(* CODESYS project ProyectoAutomatasCodesys.project

Project tree, tasks and I/O mapping:
  Device : CODESYS Control Win V3, 3S - Smart Software Solutions GmbH, order no. 305021, version 3.5.9.20
    application Application
      libraries: Standard, * (System)
      task AutomataSeguridad (cyclic, interval t#100ms, priority 4) calls Nivel0
      task AutomataSupervisor (cyclic, interval t#50ms, priority 3) calls Nivel1
      task NivelControl (cyclic, interval t#22ms, priority 2) calls nivel2prueba
      task Planta (cyclic, interval t#1ms, priority 1) calls Planta
      task VISU_TASK (cyclic, interval 100 ms, priority 31) calls VisuElems.Visu_Prg
      program Nivel2 [ST]
      function block ControlAngulo [ST]
      function block Integrador [ST]
      function block Derivador [ST]
      program Nivel0 [SFC]: DuringRestaurarFuncionamiento, DuringFuncionamientoNormal, DuringEmergencia, DuringInit_RestaurarFuncionamiento, DuringDetenerCarro, DuringRegresarCarroNormalidad, DuringCarroDentroLimites, DuringDetenerIzaje, DuringRegresarIzajeNormalidad, DuringIzajeDentroLimites
      function block PIDCarro [ST]
      function block PIDIzaje [ST]
      Symbols
      global variables Global
      program Nivel1 [SFC]: tableroDeControl_active, grua_active, maquinaEspera_active, calculoSalidas_active, manual_active, manual_entry, manual_active_0, manual_entry_0, automatico_active, habilitaControlAngulo_active, habilitado_entry, deshabilitado_entry, gancho_active, Gabierto_entry, Gcerrado_entry, Gcerrado_active, pesoPermitido_entry, manualAuto_active, automatico_entry, pesoExcedido_entry, opManual_active, carro_active, izaje_active, verificacion_active, tableroActivo_entry, tableroActivo_active, tableroActivo_entry_0, tableroActivo_exit, limitesIzaje_active, dentroDeLimites_entry, cercaMinimo_entry, cercaMaximo_entry, cercaMaximo_active, manualAuto_entry, autoManual_active, autoManual_entry, start_active, actualizarParametros_active, start_entry, barcoAlMuelle_active, subirIzaje_entry, subirYdesplazarCarro_entry, Step0_barcoAlMuelle_active_entry, bajarYdesplazarCarro_entry, bajarCarro_entry, parar_entry, parar_active, parar_exit, subirIzaje_active, subirYdesplazarCarro_active, moverCarro_active, bajarYdesplazarCarro_active, bajarCarro_active, manualAuto_exit, autoManual_exit, cercaMinimo_active, subirYdesplazar_active, generador_active
      function AjusteGananciasCarro [ST]
      function block Saturation [ST]
      function block RateLimiter [ST]
      function AjusteBordesCarro [ST]
      program Planta [ST]
      function block Carro [ST]
      function block Izaje [ST]
      function block CargaSuspendida [ST]
      function block CableElastico [ST]
      function rectaDosPuntos [ST]
      function Transferencia [ST]
      function verificarChoquesLateralesMuelle [ST]
      function verificarChoquesLateralesBarco [ST]
      function trianguloDesaceleracion [ST]
      function trianguloAceleracion [ST]
      function round [ST]
      function block GeneradorDeTrayectorias [ST]
      function colisionMuelleAlBarcoDesacel [ST]
      function colisionMuelleAlBarcoAcel [ST]
      function colisionBarcoAlMuelleDesacel [ST]
      function colisionBarcoAlMuelleAcel [ST]
      function block determinarAlturasContenedores [ST]
      visualisation Visualization
      program nivel2prueba [ST]
  libraries: VisuSymbols, 3.5.10.0 (System)
  text list GlobalTextList
*)

// Device/Application/Global
VAR_GLOBAL
	//Con la planta
	xt: LREAL :=-30;
	lh: LREAL :=5;
	theta: LREAL :=0;
	ml: LREAL :=15000;
	Tt: LREAL :=0;
	Gcierre: BOOL :=0;
	Th: LREAL :=-15000*9.80665*0.75/30;
	
	//Con el tablero y mando
	
	BotonEmergencia: BOOL:= FALSE;
	BotonReset: BOOL:= FALSE;
	BotonAbrirGancho: BOOL:= FALSE;
	BotonCerrarGancho: BOOL:= FALSE;
	BotonOperarMaq: BOOL:= FALSE;
	BotonPararMaq: BOOL:= FALSE;
	BotonModoAutomatico: BOOL:= FALSE;
	BotonModoManual: BOOL:= FALSE;
	PalancaCarro: INT:= 0;
	PalancaIzaje: INT:= 0;
	BotonActivaControlAngulo: BOOL:= FALSE;
	BotonDesactivaControlAngulo: BOOL:= FALSE;
	
	//para el generador de trayectorias
	x_destino: LREAL:= -30;
	x_origen: LREAL:= -30;
	y_destino: LREAL:= 40;
	y_origen: LREAL:= 40;
	ySeguridadCarro: LREAL:= 40;
	PosicionCarroInicioDescensoIzaje: LREAL:= -999;
	alturaInicioDesplazamientoCarro: LREAL:= -999;
	contBarco: ARRAY[1..21, 1..13] OF LREAL;
	contMuelle: ARRAY[1..2, 1..7] OF LREAL;
	//Entre nivel 0 y 1
	
	DetenerNivel1: BOOL:= FALSE;
	
	//Entre nivel 0 y 2
	
	FuncionamientoIzaje: BOOL:= TRUE;
	FuncionamientoCarro: BOOL:= TRUE;
	ConsignaCarro: LREAL:= 0;
	ConsignaIzaje: LREAL:= 0;
	
	//Entre nivel 1 y 2
	
	vh: LREAL:= 0;	
	vt: LREAL:= 0;
	ControlAngulo: BOOL:= TRUE;
	ControlPos: BOOL:= FALSE;
	
	

	//constantes que se usan en los dos niveles de control
	amaxt: LREAL:= 1;
	vmaxt: LREAL:= 4;
	amaxh: LREAL:= 1;
	vmaxh: LREAL:= 3;
	dt_control: LREAL:=0.022;
	dt_planta: LREAL:=0.001;

	
END_VAR

// Device/Application/Nivel0
PROGRAM Nivel0
VAR
	IzajeListo: BOOL:= FALSE;
	CarroListo: BOOL:= FALSE;
END_VAR
VAR CONSTANT
	l_max_max_cable: LREAL:= 66;
	l_min_min_cable: LREAL:= 4;
	xt_max_max: LREAL:= 51;
	xt_min_min: LREAL:= -31;
	l_max_cable: LREAL:= 65;
	l_min_cable: LREAL:= 5;
	xt_max: LREAL:= 50;
	xt_min: LREAL:= -30;
	vmaxh: LREAL := 3;
	vmaxt: LREAL := 4;
END_VAR

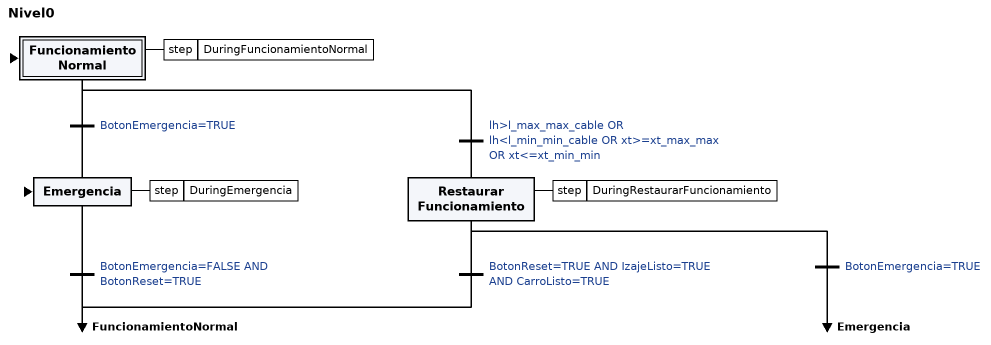
INITIAL_STEP FuncionamientoNormal:
    DuringFuncionamientoNormal(N);  // step action
END_STEP
TRANSITION FROM FuncionamientoNormal TO Emergencia
    := BotonEmergencia=TRUE;
END_TRANSITION
STEP Emergencia:
    DuringEmergencia(N);  // step action
END_STEP
TRANSITION FROM Emergencia TO FuncionamientoNormal
    := BotonEmergencia=FALSE AND BotonReset=TRUE;
END_TRANSITION
TRANSITION FROM FuncionamientoNormal TO RestaurarFuncionamiento
    := lh>l_max_max_cable OR lh<l_min_min_cable OR xt>=xt_max_max OR xt<=xt_min_min;
END_TRANSITION
STEP RestaurarFuncionamiento:
    DuringRestaurarFuncionamiento(N);  // step action
END_STEP
TRANSITION FROM RestaurarFuncionamiento TO FuncionamientoNormal
    := BotonReset=TRUE AND IzajeListo=TRUE AND CarroListo=TRUE;
END_TRANSITION
TRANSITION FROM RestaurarFuncionamiento TO Emergencia
    := BotonEmergencia=TRUE;
END_TRANSITION

ACTION DuringRestaurarFuncionamiento:
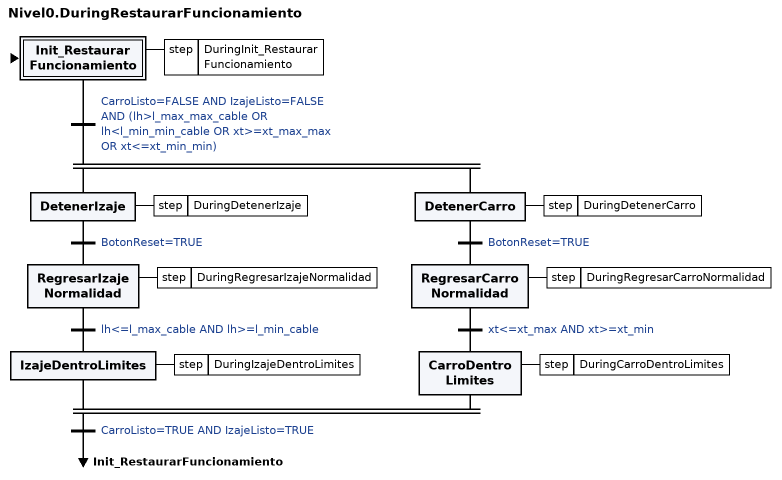
INITIAL_STEP Init_RestaurarFuncionamiento:
    DuringInit_RestaurarFuncionamiento(N);  // step action
END_STEP
TRANSITION FROM Init_RestaurarFuncionamiento TO (DetenerIzaje, DetenerCarro)
    := CarroListo=FALSE AND IzajeListo=FALSE AND (lh>l_max_max_cable OR lh<l_min_min_cable OR xt>=xt_max_max OR xt<=xt_min_min);
END_TRANSITION
STEP DetenerIzaje:
    DuringDetenerIzaje(N);  // step action
END_STEP
TRANSITION FROM DetenerIzaje TO RegresarIzajeNormalidad
    := BotonReset=TRUE;
END_TRANSITION
STEP RegresarIzajeNormalidad:
    DuringRegresarIzajeNormalidad(N);  // step action
END_STEP
TRANSITION FROM RegresarIzajeNormalidad TO IzajeDentroLimites
    := lh<=l_max_cable AND lh>=l_min_cable;
END_TRANSITION
STEP IzajeDentroLimites:
    DuringIzajeDentroLimites(N);  // step action
END_STEP
STEP DetenerCarro:
    DuringDetenerCarro(N);  // step action
END_STEP
TRANSITION FROM DetenerCarro TO RegresarCarroNormalidad
    := BotonReset=TRUE;
END_TRANSITION
STEP RegresarCarroNormalidad:
    DuringRegresarCarroNormalidad(N);  // step action
END_STEP
TRANSITION FROM RegresarCarroNormalidad TO CarroDentroLimites
    := xt<=xt_max AND xt>=xt_min;
END_TRANSITION
STEP CarroDentroLimites:
    DuringCarroDentroLimites(N);  // step action
END_STEP
TRANSITION FROM (IzajeDentroLimites, CarroDentroLimites) TO Init_RestaurarFuncionamiento
    := CarroListo=TRUE AND IzajeListo=TRUE;
END_TRANSITION
// branch label Branch0_RestaurarFuncionamiento
END_ACTION

ACTION DuringFuncionamientoNormal:
FuncionamientoIzaje:= TRUE;
FuncionamientoCarro:= TRUE;
DetenerNivel1:= FALSE;
END_ACTION

ACTION DuringEmergencia:
FuncionamientoIzaje:=FALSE;
FuncionamientoCarro:=FALSE;
ConsignaIzaje:=0;
ConsignaCarro:=0;
DetenerNivel1:=TRUE;
END_ACTION

ACTION DuringInit_RestaurarFuncionamiento:
IzajeListo:=FALSE;
CarroListo:=FALSE;
END_ACTION

ACTION DuringDetenerCarro:
IF (xt>=xt_max_max OR xt<=xt_min_min)
	THEN
	FuncionamientoCarro:= FALSE;
    ConsignaCarro:=0;
END_IF
END_ACTION

ACTION DuringRegresarCarroNormalidad:
DetenerNivel1:=TRUE;
FuncionamientoCarro:=FALSE;
IF (xt>xt_max)
	THEN
	ConsignaCarro:=-vmaxt/10;
END_IF
IF xt<xt_min
	THEN
    ConsignaCarro:=vmaxt/10;
END_IF
END_ACTION

ACTION DuringCarroDentroLimites:
CarroListo:=TRUE;
ConsignaCarro:=0;
END_ACTION

ACTION DuringDetenerIzaje:
IF (lh>l_max_max_cable OR lh<l_min_min_cable)
	THEN
	FuncionamientoIzaje:=FALSE;
    ConsignaIzaje:=0;
END_IF
END_ACTION

ACTION DuringRegresarIzajeNormalidad:
DetenerNivel1:= TRUE;
FuncionamientoIzaje:= FALSE;
IF (lh>l_max_cable)
	THEN
	ConsignaIzaje:=-vmaxh/10;
END_IF
IF (lh<l_min_cable)
	THEN
	ConsignaIzaje:=vmaxh/10;
END_IF
END_ACTION

ACTION DuringIzajeDentroLimites:
IzajeListo:=TRUE;
ConsignaIzaje:=0;
END_ACTION

END_PROGRAM

// Device/Application/Nivel1
PROGRAM Nivel1
VAR
	tiempoTableroActivo: LREAL:= 0;
	//tableroActivo:BOOL:=0;
	vhPermitidaIzq:LREAL:=0 ;
	vhPermitidaDer:LREAL:=0 ;
	finOperacion : BOOL:=1 ;
	vtmanual: LREAL := 0;
	vhmanual: LREAL := 0;
	
	vhauto: LREAL := 0;
	vtauto: LREAL := 0;
	
	x_destinoAnterior: LREAL :=999;
	Generador: GeneradorDeTrayectorias;
	
	tiempoTablero: ton ;
	tiempoManualAuto: ton ;
	tiempoModoAutomatico: ton;
	//para la transicion
	wait: ton;
	//Step: INT;
	
	//contadorTransicion: INT :=0;
	vmaxh: LREAL :=3;
	vmaxhfull: LREAL :=1.5;
	vmaxhSobrepeso: LREAL:=0.1;
	mlfull: LREAL := 65000;
	y_actual: LREAL := 45;
	//T: INT := 4;
	// auxiliar para manualAuto
	tiempo: LREAL := 0;
	cteAlturaInferior: LREAL;
	cteAlturaSuperior: LREAL;
	cteDestino: LREAL;
	n: INT := 0;
	veces: INT := 10;
	cteAlturaSuperior1: LREAL;
	cteCarro: LREAL;
END_VAR

VAR CONSTANT
	yt0: LREAL := 45;
	// se usa en limitesIzaje
	longitudSegMaxCable: LREAL := 60;
	longitudSegMinCable: LREAL := 10;
	l_max_cable: LREAL := 65;
	l_min_cable: LREAL := 5;
END_VAR

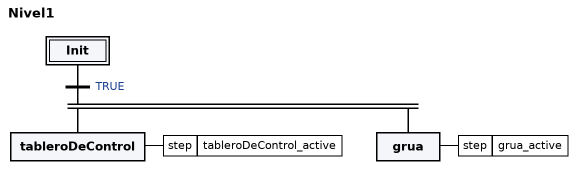
INITIAL_STEP Init:
END_STEP
TRANSITION FROM Init TO (tableroDeControl, grua)
    := TRUE;
END_TRANSITION
STEP tableroDeControl:
    tableroDeControl_active(N);  // step action
END_STEP
STEP grua:
    grua_active(N);  // step action
END_STEP

ACTION tableroDeControl_active:
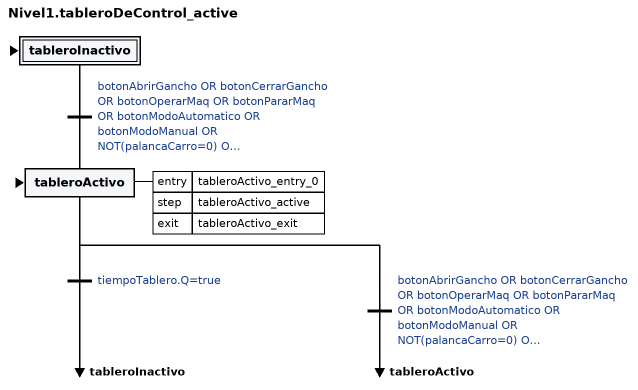
INITIAL_STEP tableroInactivo:
END_STEP
TRANSITION FROM tableroInactivo TO tableroActivo
    := botonAbrirGancho OR botonCerrarGancho OR botonOperarMaq OR botonPararMaq OR botonModoAutomatico OR botonModoManual OR NOT(palancaCarro=0) OR NOT(palancaIzaje=0);
END_TRANSITION
STEP tableroActivo:
    tableroActivo_entry_0(P1);  // entry action
    tableroActivo_active(N);  // step action
    tableroActivo_exit(P0);  // exit action
END_STEP
TRANSITION FROM tableroActivo TO tableroInactivo
    := tiempoTablero.Q=true;
END_TRANSITION
TRANSITION FROM tableroActivo TO tableroActivo
    := botonAbrirGancho OR botonCerrarGancho OR botonOperarMaq OR botonPararMaq OR botonModoAutomatico OR botonModoManual OR NOT(palancaCarro=0) OR NOT(palancaIzaje=0);
END_TRANSITION
// branch label Branch0_tableroDeControl_active
END_ACTION

ACTION grua_active:
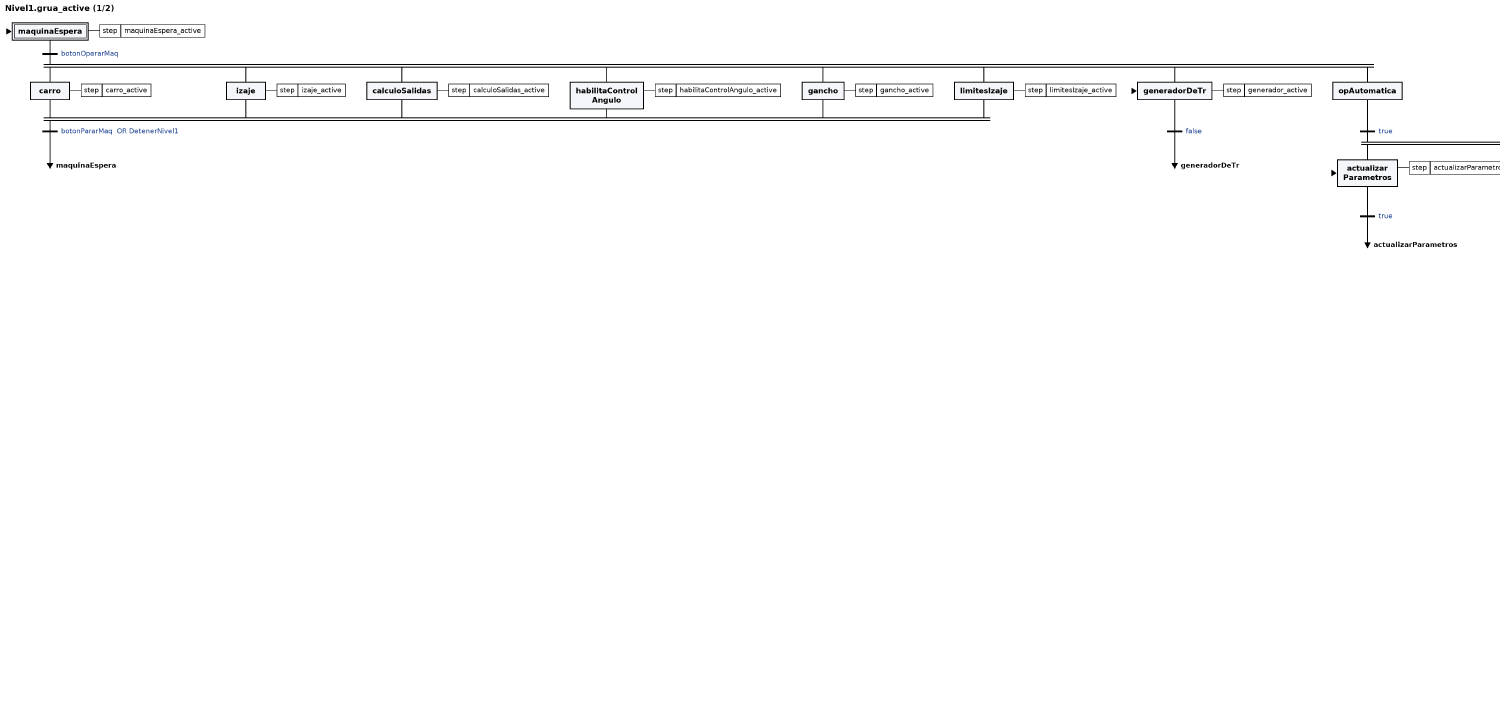
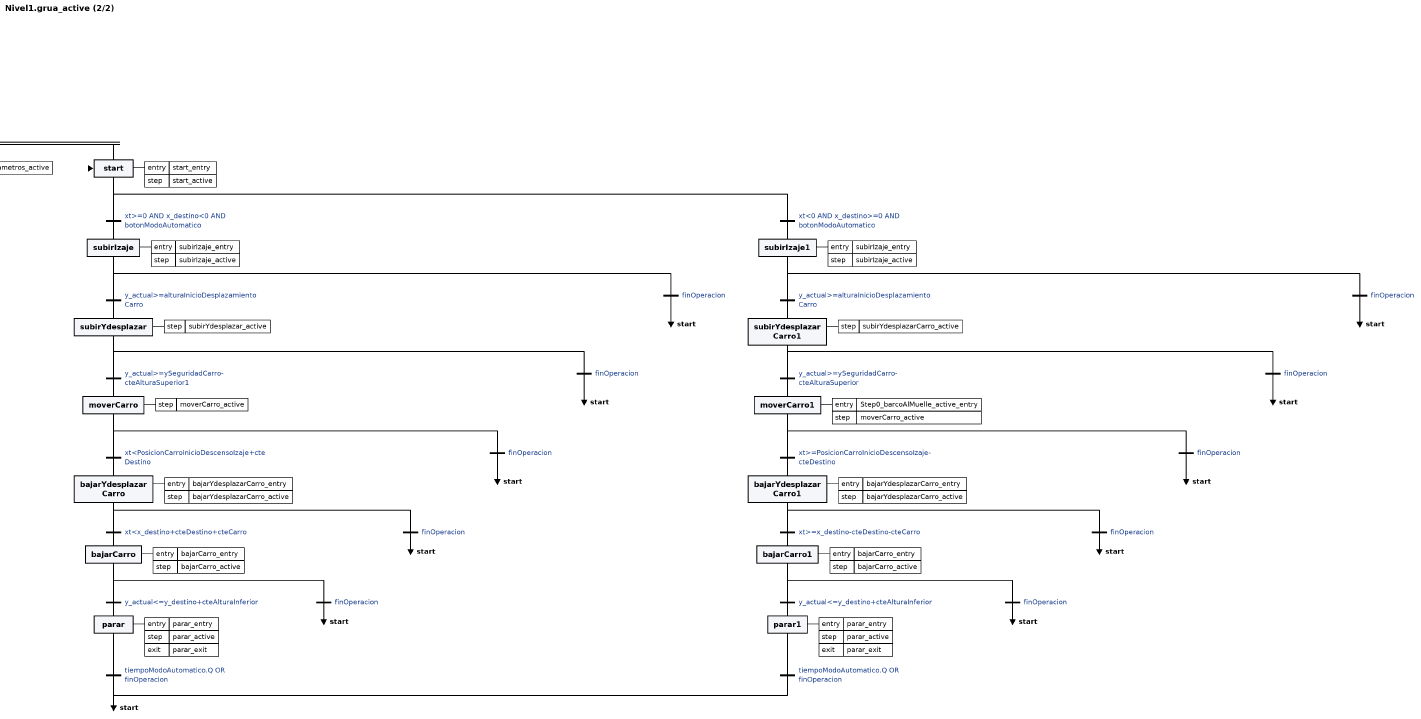
INITIAL_STEP maquinaEspera:
    maquinaEspera_active(N);  // step action
END_STEP
TRANSITION FROM maquinaEspera TO (carro, izaje, calculoSalidas, habilitaControlAngulo, gancho, limitesIzaje, generadorDeTr, opAutomatica)
    := botonOperarMaq;
END_TRANSITION
STEP carro:
    carro_active(N);  // step action
END_STEP
STEP izaje:
    izaje_active(N);  // step action
END_STEP
STEP calculoSalidas:
    calculoSalidas_active(N);  // step action
END_STEP
STEP habilitaControlAngulo:
    habilitaControlAngulo_active(N);  // step action
END_STEP
STEP gancho:
    gancho_active(N);  // step action
END_STEP
STEP limitesIzaje:
    limitesIzaje_active(N);  // step action
END_STEP
STEP generadorDeTr:
    generador_active(N);  // step action
END_STEP
TRANSITION FROM generadorDeTr TO generadorDeTr
    := false;
END_TRANSITION
STEP opAutomatica:
END_STEP
TRANSITION FROM opAutomatica TO (actualizarParametros, start)
    := true;
END_TRANSITION
STEP actualizarParametros:
    actualizarParametros_active(N);  // step action
END_STEP
TRANSITION FROM actualizarParametros TO actualizarParametros
    := true;
END_TRANSITION
STEP start:
    start_entry(P1);  // entry action
    start_active(N);  // step action
END_STEP
TRANSITION FROM start TO subirIzaje
    := xt>=0 AND x_destino<0 AND botonModoAutomatico;
END_TRANSITION
STEP subirIzaje:
    subirIzaje_entry(P1);  // entry action
    subirIzaje_active(N);  // step action
END_STEP
TRANSITION FROM subirIzaje TO subirYdesplazar
    := y_actual>=alturaInicioDesplazamientoCarro;
END_TRANSITION
STEP subirYdesplazar:
    subirYdesplazar_active(N);  // step action
END_STEP
TRANSITION FROM subirIzaje TO start
    := finOperacion;
END_TRANSITION
TRANSITION FROM subirYdesplazar TO moverCarro
    := y_actual>=ySeguridadCarro-cteAlturaSuperior1;
END_TRANSITION
TRANSITION FROM subirYdesplazar TO start
    := finOperacion;
END_TRANSITION
STEP moverCarro:
    moverCarro_active(N);  // step action
END_STEP
TRANSITION FROM moverCarro TO bajarYdesplazarCarro
    := xt<PosicionCarroInicioDescensoIzaje+cteDestino;
END_TRANSITION
TRANSITION FROM moverCarro TO start
    := finOperacion;
END_TRANSITION
STEP bajarYdesplazarCarro:
    bajarYdesplazarCarro_entry(P1);  // entry action
    bajarYdesplazarCarro_active(N);  // step action
END_STEP
TRANSITION FROM bajarYdesplazarCarro TO bajarCarro
    := xt<x_destino+cteDestino+cteCarro;
END_TRANSITION
TRANSITION FROM bajarYdesplazarCarro TO start
    := finOperacion;
END_TRANSITION
STEP bajarCarro:
    bajarCarro_entry(P1);  // entry action
    bajarCarro_active(N);  // step action
END_STEP
TRANSITION FROM bajarCarro TO parar
    := y_actual<=y_destino+cteAlturaInferior;
END_TRANSITION
TRANSITION FROM bajarCarro TO start
    := finOperacion;
END_TRANSITION
STEP parar:
    parar_entry(P1);  // entry action
    parar_active(N);  // step action
    parar_exit(P0);  // exit action
END_STEP
TRANSITION FROM parar TO start
    := tiempoModoAutomatico.Q OR finOperacion;
END_TRANSITION
TRANSITION FROM start TO subirIzaje1
    := xt<0 AND x_destino>=0 AND botonModoAutomatico;
END_TRANSITION
STEP subirIzaje1:
    subirIzaje_entry(P1);  // entry action
    subirIzaje_active(N);  // step action
END_STEP
TRANSITION FROM subirIzaje1 TO subirYdesplazarCarro1
    := y_actual>=alturaInicioDesplazamientoCarro;
END_TRANSITION
TRANSITION FROM subirIzaje1 TO start
    := finOperacion;
END_TRANSITION
STEP subirYdesplazarCarro1:
    subirYdesplazarCarro_active(N);  // step action
END_STEP
TRANSITION FROM subirYdesplazarCarro1 TO moverCarro1
    := y_actual>=ySeguridadCarro-cteAlturaSuperior;
END_TRANSITION
TRANSITION FROM subirYdesplazarCarro1 TO start
    := finOperacion;
END_TRANSITION
STEP moverCarro1:
    Step0_barcoAlMuelle_active_entry(P1);  // entry action
    moverCarro_active(N);  // step action
END_STEP
TRANSITION FROM moverCarro1 TO bajarYdesplazarCarro1
    := xt>=PosicionCarroInicioDescensoIzaje-cteDestino;
END_TRANSITION
TRANSITION FROM moverCarro1 TO start
    := finOperacion;
END_TRANSITION
STEP bajarYdesplazarCarro1:
    bajarYdesplazarCarro_entry(P1);  // entry action
    bajarYdesplazarCarro_active(N);  // step action
END_STEP
TRANSITION FROM bajarYdesplazarCarro1 TO bajarCarro1
    := xt>=x_destino-cteDestino-cteCarro;
END_TRANSITION
TRANSITION FROM bajarYdesplazarCarro1 TO start
    := finOperacion;
END_TRANSITION
STEP bajarCarro1:
    bajarCarro_entry(P1);  // entry action
    bajarCarro_active(N);  // step action
END_STEP
TRANSITION FROM bajarCarro1 TO parar1
    := y_actual<=y_destino+cteAlturaInferior;
END_TRANSITION
TRANSITION FROM bajarCarro1 TO start
    := finOperacion;
END_TRANSITION
STEP parar1:
    parar_entry(P1);  // entry action
    parar_active(N);  // step action
    parar_exit(P0);  // exit action
END_STEP
TRANSITION FROM parar1 TO start
    := tiempoModoAutomatico.Q OR finOperacion;
END_TRANSITION
TRANSITION FROM (carro, izaje, calculoSalidas, habilitaControlAngulo, gancho, limitesIzaje) TO maquinaEspera
    := botonPararMaq OR DetenerNivel1;
END_TRANSITION
// branch label Branch3_grua_active
// branch label Branch4_grua_active
// branch label Branch5_grua_active
// branch label Branch6_grua_active
// branch label Branch7_grua_active
// branch label Branch2_grua_active
// branch label Branch1_grua_active
// branch label Branch0_maquinaOperando_active
END_ACTION

ACTION maquinaEspera_active:
vt:=0;
vh:=0;
vhPermitidaIzq:=0 ;
vhPermitidaDer:=0 ;
END_ACTION

ACTION calculoSalidas_active:
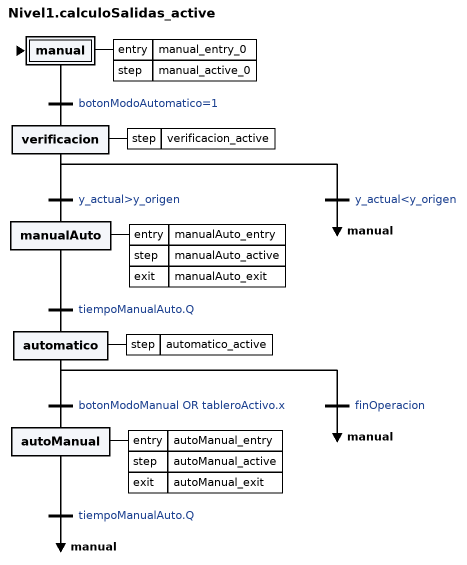
INITIAL_STEP manual:
    manual_entry_0(P1);  // entry action
    manual_active_0(N);  // step action
END_STEP
TRANSITION FROM manual TO verificacion
    := botonModoAutomatico=1;
END_TRANSITION
STEP verificacion:
    verificacion_active(N);  // step action
END_STEP
TRANSITION FROM verificacion TO manualAuto
    := y_actual>y_origen;
END_TRANSITION
TRANSITION FROM verificacion TO manual
    := y_actual<y_origen;
END_TRANSITION
STEP manualAuto:
    manualAuto_entry(P1);  // entry action
    manualAuto_active(N);  // step action
    manualAuto_exit(P0);  // exit action
END_STEP
TRANSITION FROM manualAuto TO automatico
    := tiempoManualAuto.Q;
END_TRANSITION
STEP automatico:
    automatico_active(N);  // step action
END_STEP
TRANSITION FROM automatico TO autoManual
    := botonModoManual OR tableroActivo.x;
END_TRANSITION
TRANSITION FROM automatico TO manual
    := finOperacion;
END_TRANSITION
STEP autoManual:
    autoManual_entry(P1);  // entry action
    autoManual_active(N);  // step action
    autoManual_exit(P0);  // exit action
END_STEP
TRANSITION FROM autoManual TO manual
    := tiempoManualAuto.Q;
END_TRANSITION
// branch label Branch0_calculoSalidas_active
// branch label Branch1_calculoSalidas_active
END_ACTION

ACTION manual_active:

END_ACTION

ACTION manual_entry:
controlPos :=0;
finOperacion :=1;
END_ACTION

ACTION manual_active_0:
vt :=vtmanual;
vh :=vhmanual;
END_ACTION

ACTION manual_entry_0:
controlPos :=0;
finOperacion :=1;
tiempoManualAuto.IN  :=0;
END_ACTION

ACTION automatico_active:
vt:=vtauto;
vh:=vhauto;
END_ACTION

ACTION habilitaControlAngulo_active:
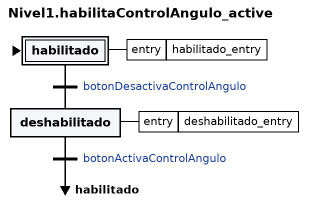
INITIAL_STEP habilitado:
    habilitado_entry(P1);  // entry action
END_STEP
TRANSITION FROM habilitado TO deshabilitado
    := botonDesactivaControlAngulo;
END_TRANSITION
STEP deshabilitado:
    deshabilitado_entry(P1);  // entry action
END_STEP
TRANSITION FROM deshabilitado TO habilitado
    := botonActivaControlAngulo;
END_TRANSITION
END_ACTION

ACTION habilitado_entry:
controlAngulo:=1;
END_ACTION

ACTION deshabilitado_entry:
controlAngulo:=0;
END_ACTION

ACTION gancho_active:
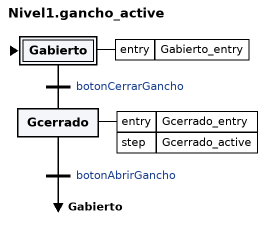
INITIAL_STEP Gabierto:
    Gabierto_entry(P1);  // entry action
END_STEP
TRANSITION FROM Gabierto TO Gcerrado
    := botonCerrarGancho;
END_TRANSITION
STEP Gcerrado:
    Gcerrado_entry(P1);  // entry action
    Gcerrado_active(N);  // step action
END_STEP
TRANSITION FROM Gcerrado TO Gabierto
    := botonAbrirGancho;
END_TRANSITION
END_ACTION

ACTION Gabierto_entry:
Gcierre:=0;
vhPermitidaIzq:=vmaxh;
vhPermitidaDer:= vmaxh;
END_ACTION

ACTION Gcerrado_entry:
Gcierre:=1;
END_ACTION

ACTION Gcerrado_active:
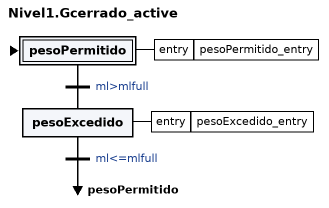
INITIAL_STEP pesoPermitido:
    pesoPermitido_entry(P1);  // entry action
END_STEP
TRANSITION FROM pesoPermitido TO pesoExcedido
    := ml>mlfull;
END_TRANSITION
STEP pesoExcedido:
    pesoExcedido_entry(P1);  // entry action
END_STEP
TRANSITION FROM pesoExcedido TO pesoPermitido
    := ml<=mlfull;
END_TRANSITION
END_ACTION

ACTION pesoPermitido_entry:
vhPermitidaIzq :=vmaxhfull ;
vhPermitidaDer:=vmaxhfull ;
END_ACTION

ACTION manualAuto_active:
tiempoManualAuto();
tiempo:=TIME_TO_LREAL(tiempoManualAuto.ET)/1000;
Transferencia(1.0,tiempo,vtmanual,vtauto,vhmanual,vhauto,Vh=>vh,Vt=>vt);
END_ACTION

ACTION automatico_entry:

END_ACTION

ACTION pesoExcedido_entry:
vhPermitidaIzq :=vmaxhSobrepeso ;
vhPermitidaDer:=vmaxhSobrepeso ;
END_ACTION

ACTION opManual_active:
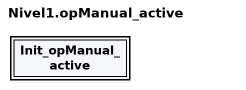
INITIAL_STEP Init_opManual_active:
END_STEP
END_ACTION

ACTION carro_active:
IF palancaCarro=-1 THEN
    vtmanual:=-vmaxt;
ELSIF palancaCarro=0 THEN
    vtmanual:=0; 
ELSIF palancaCarro=1 THEN
    vtmanual:=vmaxt;
END_IF
END_ACTION

ACTION izaje_active:
IF palancaIzaje=1 THEN
    vhmanual := vhPermitidaIzq;
ELSIF palancaIzaje=0 THEN
    vhmanual := 0;
ELSIF palancaIzaje=-1 THEN
    vhmanual := -vhPermitidaDer;
END_IF
END_ACTION

ACTION verificacion_active:
y_actual:=yt0-lh;
END_ACTION

ACTION tableroActivo_entry:
tiempoTablero(IN:=0,PT:=T#4S);
tiempoTablero.IN  :=1;
END_ACTION

ACTION tableroActivo_active:
tiempoTablero();
END_ACTION

ACTION tableroActivo_entry_0:
tiempoTablero.IN  :=0;
tiempoTablero(IN:=1,PT:=T#1S);
END_ACTION

ACTION tableroActivo_exit:
tiempoTablero(IN:=0);
END_ACTION

ACTION limitesIzaje_active:
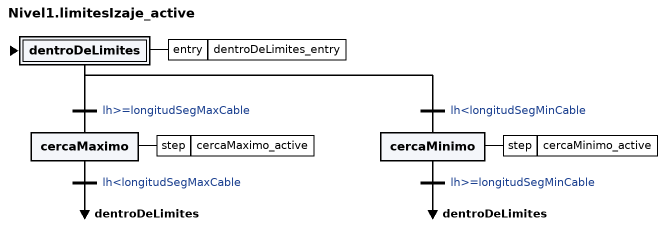
INITIAL_STEP dentroDeLimites:
    dentroDeLimites_entry(P1);  // entry action
END_STEP
TRANSITION FROM dentroDeLimites TO cercaMaximo
    := lh>=longitudSegMaxCable;
END_TRANSITION
STEP cercaMaximo:
    cercaMaximo_active(N);  // step action
END_STEP
TRANSITION FROM cercaMaximo TO dentroDeLimites
    := lh<longitudSegMaxCable;
END_TRANSITION
TRANSITION FROM dentroDeLimites TO cercaMinimo
    := lh<longitudSegMinCable;
END_TRANSITION
STEP cercaMinimo:
    cercaMinimo_active(N);  // step action
END_STEP
TRANSITION FROM cercaMinimo TO dentroDeLimites
    := lh>=longitudSegMinCable;
END_TRANSITION
// branch label Branch0_limitesIzaje_active
END_ACTION

ACTION dentroDeLimites_entry:
IF Gcierre THEN
	vhPermitidaIzq:= vmaxhfull;
	vhPermitidaDer:=vmaxhfull;
	
ELSE
	vhPermitidaIzq:=vmaxh ;
	vhPermitidaDer:=vmaxh ;
END_IF
END_ACTION

ACTION cercaMinimo_entry:

END_ACTION

ACTION cercaMaximo_entry:

END_ACTION

ACTION cercaMaximo_active:
IF Gcierre THEN
    vhPermitidaIzq:=rectaDosPuntos(vmaxh  ,0,longitudSegMaxCable,l_max_cable,lh);
else
    vhPermitidaIzq:=rectaDosPuntos(vmaxhfull,0,longitudSegMaxCable,l_max_cable,lh);
END_IF
END_ACTION

ACTION manualAuto_entry:
tiempoManualAuto.IN  :=0;
tiempoManualAuto(IN:=1,PT:=T#5S);
END_ACTION

ACTION autoManual_active:
tiempoManualAuto();
tiempo:=TIME_TO_LREAL(tiempoManualAuto.ET);
Transferencia(-1.0,tiempo,vtmanual,vtauto,vhmanual,vhauto);
END_ACTION

ACTION autoManual_entry:
tiempoManualAuto.IN  :=0;
tiempoManualAuto(IN:=1,PT:=T#5S);
END_ACTION

ACTION start_active:
y_actual:=yt0-lh;
END_ACTION

ACTION actualizarParametros_active:
 IF lh<22 THEN
     IF Gcierre THEN
         cteAlturaInferior:=6;
         cteAlturaSuperior:=-2;
         cteDestino:=0;
		 cteCarro:=10;
     else
         cteAlturaInferior:=6;
         cteAlturaSuperior:=10;
         cteDestino:=5;
		 cteCarro:=10;
     END_IF
 else
     IF Gcierre THEN
		 cteAlturaSuperior1:=2;
         cteAlturaInferior:=9;
         cteAlturaSuperior:=-2;
         cteDestino:=0;
		 cteCarro:=12;
     ELSE
		 cteAlturaSuperior1:=2;
         cteAlturaInferior:=10;
         cteAlturaSuperior:=4;
         cteDestino:=6;
		 cteCarro:=12;
     END_IF
 END_IF
END_ACTION

ACTION start_entry:
finOperacion:=0;
vtauto:=0;
vhauto:=0;
END_ACTION

ACTION barcoAlMuelle_active:
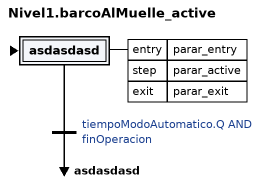
INITIAL_STEP asdasdasd:
    parar_entry(P1);  // entry action
    parar_active(N);  // step action
    parar_exit(P0);  // exit action
END_STEP
TRANSITION FROM asdasdasd TO asdasdasd
    := tiempoModoAutomatico.Q AND finOperacion;
END_TRANSITION
END_ACTION

ACTION subirIzaje_entry:

END_ACTION

ACTION subirYdesplazarCarro_entry:

END_ACTION

ACTION Step0_barcoAlMuelle_active_entry:

END_ACTION

ACTION bajarYdesplazarCarro_entry:
vhauto:=vhPermitidaIzq;
controlPos :=1;
END_ACTION

ACTION bajarCarro_entry:
vtauto:=0;
END_ACTION

ACTION parar_entry:
vhauto:=0;
tiempoModoAutomatico.IN  :=0;
tiempoModoAutomatico(IN:=1,PT:=T#60S);
END_ACTION

ACTION parar_active:
tiempoModoAutomatico();
y_actual:=yt0-lh;
END_ACTION

ACTION parar_exit:
tiempoModoAutomatico.IN  :=0;
finOperacion:=1;
END_ACTION

ACTION subirIzaje_active:
y_actual:=yt0-lh;
vhauto:=-vhPermitidaDer;
END_ACTION

ACTION subirYdesplazarCarro_active:
y_actual:=yt0-lh;
vtauto:=vmaxt;
END_ACTION

ACTION moverCarro_active:
y_actual:=yt0-lh;
vhauto:=0;
END_ACTION

ACTION bajarYdesplazarCarro_active:
y_actual:=yt0-lh;
END_ACTION

ACTION bajarCarro_active:
y_actual:=yt0-lh;
END_ACTION

ACTION manualAuto_exit:
tiempoManualAuto(IN  :=0, PT:=t#10s);
END_ACTION

ACTION autoManual_exit:
tiempoManualAuto(IN  :=0, PT:=t#10s);
END_ACTION

ACTION cercaMinimo_active:
IF Gcierre THEN
    vhPermitidaDer:=rectaDosPuntos(vmaxhfull,0,longitudSegMinCable,l_min_cable,lh);
else
    vhPermitidaDer:=rectaDosPuntos(vmaxh ,0,longitudSegMinCable,l_min_cable,lh);
END_IF
END_ACTION

ACTION subirYdesplazar_active:
y_actual:=yt0-lh;
vtauto:=-vmaxt;
END_ACTION

ACTION generador_active:
IF NOT (x_destinoAnterior=x_destino)
	THEN
	Generador();
	x_destinoAnterior:=x_destino;
END_IF
END_ACTION

END_PROGRAM

// Device/Application/GeneradorDeTrayectorias
FUNCTION_BLOCK GeneradorDeTrayectorias
VAR_INPUT
END_VAR
VAR_OUTPUT
END_VAR
VAR
	vIzaje: LREAL;
	alturaInicioAutomatico: LREAL;
	cantContDeSeguridad: LREAL;
	vCarro: LREAL;
	aTriangulo: LREAL;
	bTriangulo: LREAL;
	cTriangulo: LREAL;
	betaTriangulo: LREAL;
	determinarAlturasContenedores1: determinarAlturasContenedores;
	alturasContMuelle: ARRAY [1..7] OF LREAL;
	alturasContBarco: ARRAY [1..13] OF LREAL;
	nroColOrigen: INT;
	nroColDestino: INT;
	cuantosCont: LREAL;
	i: INT;
	donde: LREAL;
END_VAR
VAR CONSTANT
	vmaxh: LREAL:= 3;
	vmaxhfull: LREAL:= 1.5;
	vmaxt: LREAL:= 4;
	altoCont: LREAL:= 2.591;
	y_min: LREAL:=-20;
	xt_min: LREAL:= -30;
	divHoriz: LREAL:= 3.438;
	nroHorizContMuelle: INT:= 7;
	altoVigaTestera: LREAL:= 15;
	nroHorizContBarco: INT:=13;
END_VAR

//obtener posicion actual del carro
x_origen:=xt;
IF (Gcierre=1)
	THEN
    vIzaje:=vmaxhfull;
    alturaInicioAutomatico := altoCont * 1.5;
    cantContDeSeguridad:=2;
ELSE
    vIzaje:=vmaxh;
    alturaInicioAutomatico := altoCont * 0.5;
    cantContDeSeguridad:=1;
END_IF
vCarro:=vmaxt;
//calculo del triangulo de velocidades para las trayectorias
aTriangulo:=vCarro;
bTriangulo:=vIzaje;
cTriangulo:=SQRT(EXPT(aTriangulo,2)+EXPT(bTriangulo,2)); //hipotenusa
betaTriangulo:=ACOS(bTriangulo/cTriangulo);

y_destino:=999;
//inicialiar las variables, deben ser numeros negativos!!!!!!!
alturaInicioDesplazamientoCarro:=-999;
PosicionCarroInicioDescensoIzaje:=-999;
ySeguridadCarro:=-999;
//altura de seguridad para evitar colision entre el contenedor suspendido y
//las columnas de contenedores apilados. si este valor es cero, se pueden
//ver los puntos donde se encuentran los impactos.

determinarAlturasContenedores1(altoCont:= altoCont , y_min:= y_min);
alturasContMuelle:=determinarAlturasContenedores1.alturasContMuelle;
alturasContBarco:=determinarAlturasContenedores1.alturasContBarco;
//determinar si es una operacion de ida desde el barco hasta el muelle o
//viceversa
IF x_origen>=0 AND x_destino<0 //barco hasta el muelle
    THEN
    //determinar las coordenadas "Y" de las trayectorias y graficar
    nroColOrigen:=round(ABS(x_origen)/divHoriz);
    IF nroColOrigen<1
		THEN
        nroColOrigen:=1;
    END_IF
    nroColDestino:=round(ABS( (xt_min-x_destino)/divHoriz));
    y_destino:=alturasContMuelle[nroColDestino];
    cuantosCont:=2;
    y_destino:=verificarChoquesLateralesMuelle(cuantosCont:= cuantosCont, y_destino:= y_destino, nroColDestino:= nroColDestino, nroMaxCont:= nroHorizContMuelle, alturasContenedores:= alturasContMuelle, altoVigaTestera:= altoVigaTestera);
    
    //establecer la altura minima a la que debe elevarse el izaje para no chocar
    FOR i:=1 TO LREAL_TO_INT(nroColOrigen)
		DO
        IF ySeguridadCarro<alturasContBarco[i]
			THEN
            ySeguridadCarro:=alturasContBarco[i];
        END_IF
    END_FOR
    IF nroColDestino=1
		THEN
        donde:=nroColDestino;
    else
        donde:=nroColDestino-1;
    END_IF
    FOR i:=LREAL_TO_INT(donde) TO LREAL_TO_INT(nroHorizContMuelle)
		DO
        IF ySeguridadCarro<alturasContMuelle[i]
			THEN
            ySeguridadCarro:=alturasContMuelle[i];
        END_IF
    END_FOR
    IF ySeguridadCarro<=altoVigaTestera //evitar que los contenedores choquen con la viga testera
		THEN
        ySeguridadCarro:=altoVigaTestera;
    END_IF
    y_origen:=alturasContBarco[nroColOrigen];
    cuantosCont:=1;
	y_origen:=verificarChoquesLateralesBarco(cuantosCont:= cuantosCont, y_destino:= y_origen,nroColDestino:=nroColOrigen,nroMaxCont:= nroHorizContBarco, alturasContenedores:= alturasContBarco, altoVigaTestera:= AltoVigaTestera);
ELSIF x_origen<0 AND x_destino>=0 //muelle al barco
	THEN
    nroColOrigen:=round(ABS( (xt_min-x_origen)/divHoriz));
    IF nroColOrigen<1 //si la resta geometria.xt_min-x_origen es = a cero, significa que estoy en la primera columna
		THEN
        nroColOrigen:=1;
    END_IF
    nroColDestino:=DINT_TO_INT(TRUNC(ABS(x_destino)/divHoriz));
    y_destino:=alturasContBarco[nroColDestino];
    IF nroColDestino = nroHorizContBarco-1
		THEN
        IF alturasContBarco[nroHorizContBarco-1]< altoVigaTestera
			THEN
            y_destino:=altoVigaTestera; //evitar choque con la pared del barco
        END_IF
    END_IF
    cuantosCont:=2;
	y_destino:=verificarChoquesLateralesBarco(cuantosCont:=cuantosCont , y_destino:=y_destino , nroColDestino:=nroColDestino, nroMaxCont:=nroHorizContBarco , alturasContenedores:= alturasContBarco , altoVigaTestera:= altoVigaTestera);
    IF nroColDestino=1
		THEN
        IF altoVigaTestera > y_destino //si se desea llegar a la primera pila de contenedores, detenerse a la altura de la viga testera
			THEN
            y_destino:= altoVigaTestera;
        END_IF
    END_IF
    
    //establecer la altura minima a la que debe elevarse el izaje para no chocar
    IF nroColDestino<nroHorizContBarco
		THEN
        donde:=nroColDestino+1;
    ELSE
        donde:=nroColDestino;
    END_IF
    FOR i:=1 TO LREAL_TO_INT(donde)
		DO
        IF ySeguridadCarro<alturasContBarco[i]
			THEN
            ySeguridadCarro:=alturasContBarco[i];
        END_IF
    END_FOR
    FOR i:=LREAL_TO_INT(nroColOrigen) TO LREAL_TO_INT(nroHorizContMuelle)
		DO
        IF ySeguridadCarro<alturasContMuelle[i]
			THEN
            ySeguridadCarro:=alturasContMuelle[i];
        END_IF
    END_FOR
    IF ySeguridadCarro<=altoVigaTestera //evitar que los contenedores choquen con la viga testera
		THEN
        ySeguridadCarro:=altoVigaTestera;
    END_IF
    y_origen:=alturasContMuelle[nroColOrigen];
    cuantosCont:=1;
	y_origen:=verificarChoquesLateralesMuelle(cuantosCont:= cuantosCont, y_destino:= y_origen, nroColDestino:= nroColOrigen, nroMaxCont:= nroHorizContMuelle, alturasContenedores:= alturasContMuelle, altoVigaTestera:= altoVigaTestera);
END_IF

ySeguridadCarro:=ySeguridadCarro+cantContDeSeguridad*altoCont; //el sistema pasara siempre a una altura equivalente a dos contenedores cuando se desplace
y_origen := y_origen + alturaInicioAutomatico;
IF y_origen>ySeguridadCarro
	THEN
    ySeguridadCarro:=y_origen;
END_IF

alturaInicioDesplazamientoCarro:=trianguloAceleracion(ySeguridadCarro,x_origen,y_origen,betaTriangulo,nroColOrigen,alturasContBarco,alturasContMuelle,cantContDeSeguridad,altoCont);
PosicionCarroInicioDescensoIzaje:=trianguloDesaceleracion(ySeguridadCarro,x_origen,x_destino,y_destino,betaTriangulo,nroColDestino,alturasContBarco,alturasContMuelle,cantContDeSeguridad,altoCont);

END_FUNCTION_BLOCK

// Device/Application/Carro
FUNCTION_BLOCK Carro
VAR_INPUT
	SenoCarga : LREAL;
	Fw : LREAL;
	T : LREAL;
END_VAR
VAR_OUTPUT
	x : LREAL:=-30;
END_VAR
VAR
	Integrador1: Integrador;
	Integrador2: Integrador;
	init: BOOL:= FALSE;
END_VAR
VAR CONSTANT
	Mt_1: LREAL:= 1.694685466377440E-05;
	bt: LREAL:= 27000;
	rc_Rw: LREAL:= 30;
END_VAR

IF (init=FALSE)	THEN
	Integrador2(ValorActual:=-30/dt_planta,Paso:=dt_planta);
	init:=TRUE;
END_IF
Integrador1(ValorActual:= (Fw*SenoCarga+T*rc_Rw-bt*Integrador1.Integral)*Mt_1,Paso:=dt_planta);
Integrador2(ValorActual:= Integrador1.Integral,Paso:=dt_planta);
x:= Integrador2.Integral;

END_FUNCTION_BLOCK

// Device/Application/Integrador
FUNCTION_BLOCK Integrador
VAR_INPUT
	ValorActual: LREAL:= 0;
	Paso: LREAL;//:=0.001;
END_VAR
VAR_OUTPUT
	Integral: LREAL;
END_VAR
VAR
	IntegralAnterior: LREAL:= 0;
END_VAR

Integral:= IntegralAnterior+ValorActual*Paso;
IntegralAnterior:=Integral;

END_FUNCTION_BLOCK

// Device/Application/round
FUNCTION round : int
VAR_INPUT
	Imput: LREAL;
END_VAR
VAR
END_VAR

round:=LREAL_TO_INT(Imput);

END_FUNCTION

// Device/Application/verificarChoquesLateralesMuelle
FUNCTION verificarChoquesLateralesMuelle : LREAL
VAR_INPUT
	cuantosCont: LREAL;
	y_destino: LREAL;
	nroColDestino: LREAL;
	nroMaxCont: int;
	alturasContenedores: ARRAY [1..7] OF LREAL;;
	altoVigaTestera: LREAL;
END_VAR
VAR
	inicio: LREAL;
	fin: LREAL;
	i: INT;
END_VAR

//verificar si a cada lado del destino la pila de contenedores es mas
//alta, de ser asi, modificar el valor de la y_destino para evitar choques
//laterales debido a las oscilaciones
//se sube la y_destino hasta la altura de dos columnas de contenedores a
//cada lado
IF nroColDestino=1
	THEN
    inicio:=1;
    fin:=nroColDestino+cuantosCont;
ELSIF nroColDestino=2
	THEN
    inicio:=1;
    fin:=nroColDestino+cuantosCont;
ELSIF nroColDestino=nroMaxCont-1
	THEN
    inicio := nroColDestino -cuantosCont;
    fin:=nroColDestino+1;
ELSIF nroColDestino=nroMaxCont //esta en la ultima columna
	THEN
    inicio := nroColDestino -cuantosCont;
    fin :=nroColDestino;
    IF alturasContenedores[nroMaxCont]< altoVigaTestera
		THEN
        y_destino:=altoVigaTestera; //evitar choque con la pared del barco
    END_IF 
ELSE //esta en cualquier posicion intermedia
    inicio := nroColDestino - cuantosCont;
    fin:=nroColDestino + cuantosCont;
END_IF
FOR i:=LREAL_TO_INT(inicio) TO LREAL_TO_INT(fin)
	DO
    IF NOT(nroColDestino=i)
		THEN
        IF alturasContenedores[i] > y_destino //al lado es mas alto
			THEN
            y_destino:=alturasContenedores[i];
        END_IF
    END_IF
END_FOR
verificarChoquesLateralesMuelle:=y_destino;

END_FUNCTION

// Device/Application/Izaje
FUNCTION_BLOCK Izaje
VAR_INPUT
	Fw : LREAL;
	T : LREAL;
END_VAR
VAR_OUTPUT
	Lh : LREAL:=5;
	vl : LREAL:=0;
END_VAR
VAR
	Integrador1: Integrador;
	Integrador2: Integrador;
	init: BOOL:= FALSE;
END_VAR
VAR CONSTANT
	Mh_1: LREAL:= 2.082716232227488E-05;
	bh: LREAL:= 28800;
	rh_Rd: LREAL:= -40;
END_VAR

IF (init=FALSE)
	THEN
	Integrador2(ValorActual:=5/dt_planta,Paso:=dt_planta);
	init:=TRUE;
END_IF
Integrador1(ValorActual:= (Fw-T*rh_Rd-bh*Integrador1.Integral)*Mh_1,Paso:=dt_planta);
Integrador2(ValorActual:= Integrador1.Integral,Paso:=dt_planta);
Lh:= Integrador2.Integral;
vl:= Integrador1.Integral;

END_FUNCTION_BLOCK

// Device/Application/verificarChoquesLateralesBarco
FUNCTION verificarChoquesLateralesBarco : LREAL
VAR_INPUT
	cuantosCont: LREAL;
	y_destino: LREAL;
	nroColDestino: LREAL;
	nroMaxCont: INT;
	alturasContenedores: ARRAY [1..13] OF LREAL;;
	altoVigaTestera: LREAL;
END_VAR
VAR
	inicio: LREAL;
	fin: LREAL;
	i: INT;
END_VAR

//verificar si a cada lado del destino la pila de contenedores es mas
//alta, de ser asi, modificar el valor de la y_destino para evitar choques
//laterales debido a las oscilaciones
//se sube la y_destino hasta la altura de dos columnas de contenedores a
//cada lado
IF nroColDestino=1
	THEN
    inicio:=1;
    fin:=nroColDestino+cuantosCont;
ELSIF nroColDestino=2
	THEN
    inicio:=1;
    fin:=nroColDestino+cuantosCont;
ELSIF nroColDestino=nroMaxCont-1
	THEN
    inicio := nroColDestino -cuantosCont;
    fin:=nroColDestino+1;
ELSIF nroColDestino=nroMaxCont //esta en la ultima columna
	THEN
    inicio := nroColDestino -cuantosCont;
    fin :=nroColDestino;
    IF alturasContenedores[nroMaxCont]< altoVigaTestera
		THEN
        y_destino:=altoVigaTestera; //evitar choque con la pared del barco
    END_IF 
ELSE //esta en cualquier posicion intermedia
    inicio := nroColDestino - cuantosCont;
    fin:=nroColDestino + cuantosCont;
END_IF
FOR i:=LREAL_TO_INT(inicio) TO LREAL_TO_INT(fin)
	DO
    IF NOT(nroColDestino=i)
		THEN
        IF alturasContenedores[i] > y_destino //al lado es mas alto
			THEN
            y_destino:=alturasContenedores[i];
        END_IF
    END_IF
END_FOR
verificarChoquesLateralesBarco:=y_destino;

END_FUNCTION

// Device/Application/trianguloAceleracion
FUNCTION trianguloAceleracion : LREAL
VAR_INPUT
	ySeguridadCarro: LREAL;
	x_origen: LREAL;
	y_origen: LREAL;
	betaTriangulo: LREAL;
	nroColOrigen: INT;
	alturasContBarco: ARRAY [1..13] OF LREAL;
	alturasContMuelle: ARRAY [1..7] OF LREAL;
	cantContDeSeguridad: LREAL;
	altoCont: LREAL;
END_VAR
VAR
	deltaAltura: LREAL;
	catetoVert: LREAL;
	catetoHoriz: LREAL;
	i: INT;
	salida: BOOL:= 0;
END_VAR
VAR CONSTANT
	altoVigaTestera: LREAL:= 15;
END_VAR

//encontrar la altura minima a la que el carro puede comenzar a moverse sin
//chocar contenedores que puedan haber debajo de la altura de seguridad
//para esto se va descendiendo de a poco y buscando con una linea de angulo
//beta si hay contenedores en la trayectoria. al encontrar un impacto se
//detiene la busqueda
// los valores de catetoVert y catetoHoriz se utilizan para determinar la alturaInicioDesplazamientoCarro

deltaAltura:=1; //desciende de a 1 metro y evalua colisiones
IF ((ySeguridadCarro-y_origen)<INT_TO_LREAL(LREAL_TO_INT(ySeguridadCarro)-LREAL_TO_INT(y_origen)))
	THEN
	y_origen:=y_origen+1; //compensamos el error de aproximacion
END_IF

IF x_origen>0 //barco hacia el muelle  %TODO: esta condicion ya se verifico en la funcion calcularPuntosInicioMovimiento, codigo duplicado!!!
	THEN
    //     y_origen=alturasContBarco(nroColOrigen);
    
    //descender desde la altura maxima hasta donde esta el contenedor a mover
    FOR i:=LREAL_TO_INT(ySeguridadCarro) TO LREAL_TO_INT(y_origen) BY LREAL_TO_INT(-deltaAltura)    //for i=ySeguridadCarro:-geometria.altoCont:y_origen
		DO
        catetoVert:= ySeguridadCarro-(i+ySeguridadCarro-LREAL_TO_INT(ySeguridadCarro));            //geometria.altoCont*( (ySeguridadCarro-i)/geometria.altoCont );
        catetoHoriz:=TAN(betaTriangulo)*catetoVert;
        IF colisionBarcoAlMuelleAcel(catetoHoriz:=catetoHoriz , ySeguridadCarro:=ySeguridadCarro , betatriangulo:=betatriangulo , x_origen:=x_origen , nroColOrigen:=nroColOrigen , alturasContBarco:=AlturasContBarco , alturasContMuelle:= AlturasContMuelle , AltoVigaTestera:=AltoVigaTestera)
            THEN
			salida:=1;
			EXIT;
			END_IF
     END_FOR
ELSE //desde el muelle hacia el barco
    //     y_origen=alturasContMuelle(nroColOrigen);
    
    //descender desde la altura maxima hasta donde esta el contenedor a mover
    FOR i:=LREAL_TO_INT(ySeguridadCarro) TO LREAL_TO_INT(y_origen) BY LREAL_TO_INT(-deltaAltura)    //for i=ySeguridadCarro:-geometria.altoCont:y_origen
		DO
        catetoVert:= ySeguridadCarro-(i+ySeguridadCarro-LREAL_TO_INT(ySeguridadCarro));      //geometria.altoCont*( (ySeguridadCarro-i)/geometria.altoCont );
        catetoHoriz:=TAN(betaTriangulo)*catetoVert;
		IF colisionMuelleAlBarcoAcel(catetoHoriz,ySeguridadCarro,betaTriangulo,x_origen,nroColOrigen,alturasContMuelle,alturasContBarco,altoVigaTestera)
            THEN
			salida:=1;
			EXIT;
		END_IF
    END_FOR
END_IF //muelle al barco


//dar una altura mayor para evitar colision entre el contenedor transportado
//y las columnas apiladas
IF NOT salida
	THEN
	i:=i+1;
END_IF

IF ((ySeguridadCarro-(i+ySeguridadCarro-LREAL_TO_INT(ySeguridadCarro))*deltaAltura)/altoCont)-cantContDeSeguridad >0.01
	THEN
    catetoVert:=altoCont*( ((ySeguridadCarro-(i+ySeguridadCarro-LREAL_TO_INT(ySeguridadCarro))*deltaAltura)/altoCont)-cantContDeSeguridad );
    catetoHoriz:=(SIN(betaTriangulo)*catetoVert)/COS(betaTriangulo);
    alturaInicioDesplazamientoCarro:=ySeguridadCarro-catetoVert;
ELSE //ascenso primero, luego mover el carro, ambos movimientos separados
    alturaInicioDesplazamientoCarro:=ySeguridadCarro;
END_IF
trianguloAceleracion:= alturaInicioDesplazamientoCarro;

END_FUNCTION

// Device/Application/colisionBarcoAlMuelleAcel
FUNCTION colisionBarcoAlMuelleAcel : bool
VAR_INPUT
	catetoHoriz :LREAL;
	ySeguridadCarro :LREAL;
	betaTriangulo :LREAL;
	x_origen :LREAL;
	nroColOrigen :INT;
	alturasContBarco: ARRAY [1..13] OF LREAL;
	alturasContMuelle: ARRAY [1..7] OF LREAL;
	AltoVigaTestera :LREAL;
END_VAR
VAR
	detener: BOOL;
	coordxTriangulo: LREAL;
	nroColActual: INT;
	iterador: LREAL;
	k: INT;
	cuantasColumnas: LREAL;
	distHoriz: LREAL;
	distVertTrayectoria: LREAL;
	columnaCorresponde: int;
END_VAR
VAR CONSTANT
	divHoriz: LREAL:= 3.438;
	nroHorizContMuelle: INT:=7;
	xt_min: LREAL:=-30;
END_VAR

//nroColOrigen es el nroColDestino, se usan los mismos nombres de variables que en trianguloAceleracion
//x_origen puede ser x_origen o x_origen, se usan los mismo nombres que en la funcion de colisionMuelleAlBarco

detener:=FALSE;


if x_origen >=0
	THEN
    coordxTriangulo:=x_origen-catetoHoriz;
    nroColActual:=DINT_TO_INT(TRUNC(coordxTriangulo/divHoriz));
    iterador:=1;
    FOR k:=nroColActual TO nroColOrigen
		DO
        //verificar colisiones sobre el barco
        IF k>=1
			THEN
            //determinar la altura por donde pasaria la trayectoria
            cuantasColumnas:=nroColOrigen-k;
            distHoriz:=catetoHoriz-cuantasColumnas*divHoriz;
            distVertTrayectoria:=distHoriz/TAN(betaTriangulo);
            IF alturasContBarco[k] > (ySeguridadCarro-distVertTrayectoria) //si la altura de la columna de contenedores es mayor que la trayectoria sobre la misma
                THEN
				detener:=1;
                EXIT;
            END_IF
            //verificar colisiones sobre el muelle y viga testera
        else
            //determinar la altura por donde pasaria la trayectoria
            cuantasColumnas:=nroColOrigen-k;
            distHoriz:=catetoHoriz-cuantasColumnas*divHoriz;
            IF distHoriz<0
				THEN
                distHoriz:=0;//poner el break aca????
            END_IF
            distVertTrayectoria:=distHoriz/TAN(betaTriangulo);
            //viga testera
            IF altoVigaTestera > (ySeguridadCarro-distVertTrayectoria) AND coordxTriangulo<=0 //TODO: verificar si esta bien este condicional, si es coherente
				THEN
                detener:=1;
                EXIT;
            END_IF
            //muelle
            IF coordxTriangulo<=(nroHorizContMuelle+1)*divHoriz+xt_min //efectivamente la trayectoria pasa sobre los contenedores del muelle
                THEN
				columnaCorresponde:=nroHorizContMuelle+k;
                IF columnaCorresponde<=0
					THEN
                    detener:=1;
                    EXIT;
                ELSIF alturasContMuelle[columnaCorresponde] > (ySeguridadCarro-distVertTrayectoria)
					THEN
                    detener:=1;
                    EXIT;
                END_IF
            END_IF
        END_IF
    END_FOR
END_IF
colisionBarcoAlMuelleAcel:= detener;

END_FUNCTION

// Device/Application/colisionMuelleAlBarcoAcel
FUNCTION colisionMuelleAlBarcoAcel : bool
VAR_INPUT
	catetoHoriz: LREAL;
	ySeguridadCarro: LREAL;
	betaTriangulo: LREAL;
	x_origen: LREAL;
	nroColOrigen: INT;
	alturasContMuelle: ARRAY [1..7] OF LREAL;
	alturasContBarco: ARRAY [1..13] OF LREAL;
	altoVigaTestera: LREAL;
END_VAR
VAR
	detener: BOOL;
	coordxTriangulo: LREAL;
	nroColActual: INT;
	k: INT;
	cuantasColumnas: LREAL;
	distHoriz: LREAL;
	distVertTrayectoria: LREAL;
	columnaCorresponde: INT;
END_VAR
VAR CONSTANT
	divHoriz: LREAL:= 3.438;
	nroHorizContMuelle: INT:=7;
	separacionEntreCont: LREAL:= 1;
	nroHorizContBarco: LREAL:= 13;
END_VAR

//nroColOrigen es el nroColDestino, se usan los mismos nombres de variables que en trianguloAceleracion
//x_origen puede ser x_origen o x_destino, se usan los mismo nombres que en la funcion de colisionMuelleAlBarco

detener:=0;

coordxTriangulo:=x_origen+catetoHoriz;
nroColActual:=nroColOrigen + DINT_TO_INT(TRUNC(ABS( (x_origen-coordxTriangulo)/divHoriz  )));
// iterador=1;

//TODO: este codigo es exactamente igual que colisionBarcoAlMuelleDesacel

FOR k:=nroColOrigen TO nroColActual
	DO
    //verificar colisiones sobre el muelle
    IF k<=nroHorizContMuelle
		THEN
        //determinar la altura por donde pasaria la trayectoria
        cuantasColumnas:=k;
        distHoriz:=catetoHoriz-cuantasColumnas*divHoriz;
        distVertTrayectoria:=distHoriz/TAN(betaTriangulo);
        IF alturasContMuelle[k] > (ySeguridadCarro-distVertTrayectoria) //si la altura de la columna de contenedores es mayor que la trayectoria sobre la misma
			THEN
            detener:=1;
            EXIT;
        END_IF
        
        
        //verificar colisiones sobre el barco y viga testera
    else
        
        //determinar la altura por donde pasaria la trayectoria
        cuantasColumnas:=k;
        distHoriz:=catetoHoriz-cuantasColumnas*divHoriz+20;
        IF distHoriz<0
			THEN
            distHoriz:=0;//poner el break aca????
        END_IF
        distVertTrayectoria:=distHoriz/TAN(betaTriangulo);
        //viga testera
        IF altoVigaTestera > (ySeguridadCarro-distVertTrayectoria) AND coordxTriangulo>=0 //TODO: verificar si esta bien este condicional, si es coherente
			THEN
            detener:=1;
            EXIT;
        END_IF
        IF coordxTriangulo>separacionEntreCont //efectivamente la trayectoria pasa sobre los contenedores del barco
			THEN
            columnaCorresponde:=k-nroHorizContMuelle;
            IF columnaCorresponde=0
				THEN
                columnaCorresponde:=1;
            END_IF
            IF columnaCorresponde> nroHorizContBarco
				THEN
                detener:=1;
                EXIT;
            ELSIF alturasContBarco[columnaCorresponde] > (ySeguridadCarro-distVertTrayectoria)
				THEN
                detener:=1;
                EXIT;
            END_IF
        END_IF
    END_IF
END_FOR
colisionMuelleAlBarcoAcel:=detener;

END_FUNCTION

// Device/Application/colisionBarcoAlMuelleDesacel
FUNCTION colisionBarcoAlMuelleDesacel : BOOL
VAR_INPUT
catetoHoriz: LREAL;
ySeguridadCarro: LREAL;
betaTriangulo: LREAL;
x_origen: LREAL;
nroColOrigen: INT;
alturasContBarco: ARRAY[1..13] OF LREAL;
alturasContMuelle: ARRAY[1..7] OF LREAL;
END_VAR
VAR
	detener: BOOL;
	coordxTriangulo: LREAL;
	nroColActual: INT;
	k: INT;
	cuantasColumnas: INT;
	distHoriz: LREAL;
	distVertTrayectoria: LREAL;
	columnaCorresponde: INT;
END_VAR
VAR CONSTANT
	divHoriz: LREAL:= 3.438;
	nroHorizContMuelle: INT:= 7;
	altoVigaTestera: LREAL:= 15;
	separacionEntreCont: LREAL:= 1;
	nroHorizContBarco: LREAL:=13;
END_VAR

//nroColOrigen es el nroColDestino, se usan los mismos nombres de variables que en trianguloAceleracion
//x_origen puede ser x_origen o x_destino, se usan los mismo nombres que en la funcion de colisionMuelleAlBarco


//TODO: verificar que la x_origen no este antes de la posicion actual del
//carro y hacer detener=1

detener:=0;

IF x_origen <0    //hay que desacelerar sobre el muelle
	THEN
    detener:=0;
	coordxTriangulo:=x_origen+catetoHoriz;
	nroColActual:=nroColOrigen + DINT_TO_INT(TRUNC(ABS( (x_origen-coordxTriangulo)/divHoriz)));
//TODO: este codigo es exactamente igual que colisionBarcoAlMuelleDesacel

	FOR k:=nroColOrigen TO nroColActual
    //determinar la altura por donde pasaria la trayectoria
	DO
    //verificar colisiones sobre el muelle
    IF k<=nroHorizContMuelle
		THEN
        //determinar la altura por donde pasaria la trayectoria
        cuantasColumnas:=k;//nroColOrigen-k;
        distHoriz:=catetoHoriz-cuantasColumnas*divHoriz;
        distVertTrayectoria:=distHoriz/TAN(betaTriangulo);
        IF alturasContMuelle[k] > (ySeguridadCarro-distVertTrayectoria) //si la altura de la columna de contenedores es mayor que la trayectoria sobre la misma
			THEN
            detener:=1;
            EXIT;
        END_IF
        
        
        //verificar colisiones sobre el barco y viga testera
    else
        
        //determinar la altura por donde pasaria la trayectoria
        cuantasColumnas:=k;
        distHoriz:=catetoHoriz-cuantasColumnas*divHoriz+20;
        IF distHoriz<0
			THEN
            distHoriz:=0;//poner el break aca????
        END_IF
        distVertTrayectoria:=distHoriz/TAN(betaTriangulo);
        //viga testera
        IF altoVigaTestera > (ySeguridadCarro-distVertTrayectoria) AND coordxTriangulo>=0 //TODO: verificar si esta bien este condicional, si es coherente
			THEN
            detener:=1;
            EXIT;
        END_IF
        //         %barco

        IF coordxTriangulo>separacionEntreCont //efectivamente la trayectoria pasa sobre los contenedores del barco
			THEN
            columnaCorresponde:=k-nroHorizContMuelle;
            IF columnaCorresponde=0
				THEN
                columnaCorresponde:=1;
            END_IF
            IF columnaCorresponde> nroHorizContBarco
				THEN
                detener:=1;
                EXIT;
            ELSIF alturasContBarco[columnaCorresponde] > (ySeguridadCarro-distVertTrayectoria)
				THEN
                detener:=1;
                EXIT;
            END_IF
        END_IF
        
        
    END_IF
	END_FOR
    
END_IF
colisionBarcoAlMuelleDesacel:=detener;

END_FUNCTION

// Device/Application/trianguloDesaceleracion
FUNCTION trianguloDesaceleracion : LREAL
VAR_INPUT
	ySeguridadCarro: LREAL;
	x_origen: LREAL;
	x_destino: LREAL;
	y_origen: LREAL;
	betaTriangulo: LREAL;
	nroColOrigen: INT;
	alturasContBarco: ARRAY[1..13] OF LREAL;
	alturasContMuelle: ARRAY[1..7] OF LREAL;
	contenedoresDeSeguridad: LREAL;
	altoCont: LREAL;
END_VAR
VAR
	deltaAltura: LREAL;
	catetoVert: LREAL;
	catetoHoriz: LREAL;
	i: INT;
	coordxTriangulo: LREAL;
	salida: BOOL:= 0;
END_VAR
VAR CONSTANT
	divHoriz: LREAL:= 3.438;
	xt_min: LREAL:=-30;
END_VAR

//encontrar el lugar de la trayectoria del carro donde el izaje puede comenzar a descender para evitar colisiones con contenedores que puedan haber debajo de la altura de seguridad
//nroColOrigen es el nroColDestino, se usan los mismos nombres de variables que en trianguloAceleracion
//y_origen es y_destino, se usan los mismos nombres de variables

deltaAltura:=1; //desciende de a 1 metro y evalua colisiones
IF ((ySeguridadCarro-y_origen)<INT_TO_LREAL(LREAL_TO_INT(ySeguridadCarro)-LREAL_TO_INT(y_origen)))
	THEN
	y_origen:=y_origen+1; //compensamos el error de aproximacion
END_IF
if x_destino<0  //x_origen>0 %barco hacia el muelle  %TODO: esta condicion ya se verifico en la funcion calcularPuntosInicioMovimiento, codigo duplicado!!!
    //descender desde la altura maxima hasta donde esta el contenedor a mover
	THEN
    FOR i:=LREAL_TO_INT(ySeguridadCarro) TO LREAL_TO_INT(y_origen) BY LREAL_TO_INT(-deltaAltura)
		do
        catetoVert:=altoCont*( (ySeguridadCarro-(i+ySeguridadCarro-LREAL_TO_INT(ySeguridadCarro))*deltaAltura)/altoCont );
        catetoHoriz:=tan(betaTriangulo)*catetoVert;
        coordxTriangulo:=x_destino+catetoHoriz;
        if coordxTriangulo > x_origen+5
			THEN
			salida:=1;
            exit;
        end_if
        IF colisionBarcoAlMuelleDesacel(CatetoHoriz,ySeguridadCarro,betaTriangulo,x_destino,nroColOrigen,alturasContBarco,alturasContMuelle)
			THEN
			salida:=1;
            exit;
        end_if
        
    end_for
else //desde el muelle hacia el barco
    //descender desde la altura maxima hasta donde esta el contenedor a mover
    FOR i:=LREAL_TO_INT(ySeguridadCarro) TO LREAL_TO_INT(y_origen) BY LREAL_TO_INT(-deltaAltura)
		do
        catetoVert:=altoCont*( (ySeguridadCarro-(i+ySeguridadCarro-LREAL_TO_INT(ySeguridadCarro))*deltaAltura)/altoCont );
        catetoHoriz:=TAN(betaTriangulo)*catetoVert;
        IF colisionMuelleAlBarcoDesacel(catetoHoriz,ySeguridadCarro,betaTriangulo,x_destino,nroColOrigen,alturasContBarco,alturasContMuelle)
			THEN
			salida:=1;
            exit;
        end_if
    end_for
END_IF //muelle al barco
IF NOT salida
	THEN
	i:=i+1;
END_IF

IF ((ySeguridadCarro-(i+ySeguridadCarro-LREAL_TO_INT(ySeguridadCarro))*deltaAltura)/altoCont)-contenedoresDeSeguridad >0.01 //usando 0.01 se evitan errores numericos
	THEN
    catetoVert:=altoCont*( ((ySeguridadCarro-(i+ySeguridadCarro-LREAL_TO_INT(ySeguridadCarro))*deltaAltura)/altoCont)-contenedoresDeSeguridad );
    catetoHoriz:=(SIN(betaTriangulo)*catetoVert)/COS(betaTriangulo);
    
    IF x_destino<0 //se parte del barco hacia el muelle
		THEN
        PosicionCarroInicioDescensoIzaje:=nroColOrigen*divHoriz+xt_min+catetoHoriz;
    else //se parte desde el muelle hacia el barco
        PosicionCarroInicioDescensoIzaje:=nroColOrigen*divHoriz-catetoHoriz; //nroColOrigen es el nroColDestino
    end_if
else //ascenso primero, luego mover el carro, ambos movimientos separados
    PosicionCarroInicioDescensoIzaje:=x_destino;
end_if
trianguloDesaceleracion:=PosicionCarroInicioDescensoIzaje-20;

END_FUNCTION

// Device/Application/colisionMuelleAlBarcoDesacel
FUNCTION colisionMuelleAlBarcoDesacel : bool
VAR_INPUT
catetoHoriz: LREAL;
ySeguridadCarro: LREAL;
betaTriangulo: LREAL;
x_origen: LREAL;
nroColOrigen: INT;
alturasContBarco: ARRAY[1..13] OF LREAL;
alturasContMuelle: ARRAY[1..7] OF LREAL;
END_VAR
VAR
	detener: BOOL;
	coordxTriangulo: LREAL;
	nroColActual: INT;
	k: INT;
	cuantasColumnas: INT;
	distHoriz: LREAL;
	distVertTrayectoria: LREAL;
	columnaCorresponde: INT;
END_VAR
VAR CONSTANT
	divHoriz: LREAL:= 3.438;
	nroHorizContMuelle: int:= 7;
	altoVigaTestera: LREAL:= 15;
	separacionEntreCont: LREAL:= 1;
	nroHorizContBarco: LREAL:=13;
	xt_min: LREAL:=-30;
END_VAR

detener:=0;

coordxTriangulo:=x_destino-catetoHoriz;
nroColActual:=DINT_TO_INT(TRUNC(coordxTriangulo/divHoriz));

FOR k:=nroColActual TO nroColOrigen
	DO
    IF k>=1
		THEN
        //determinar la altura por donde pasaria la trayectoria
        cuantasColumnas:=nroColOrigen-k;
        distHoriz:=catetoHoriz-cuantasColumnas*divHoriz;
        distVertTrayectoria:=distHoriz/TAN(betaTriangulo);
        IF alturasContBarco[k] > (ySeguridadCarro-distVertTrayectoria) //si la altura de la columna de contenedores es mayor que la trayectoria sobre la misma
			THEN
            detener:=1;
            EXIT;
        END_IF
    ELSE
        //determinar la altura por donde pasaria la trayectoria
        cuantasColumnas:=nroColOrigen-k;
        distHoriz:=catetoHoriz-cuantasColumnas*divHoriz;
        IF distHoriz<0
			THEN
            distHoriz:=0;//poner el break aca????
        END_IF
        distVertTrayectoria:=distHoriz/TAN(betaTriangulo);
        //viga testera
        IF altoVigaTestera > (ySeguridadCarro-distVertTrayectoria) AND coordxTriangulo<=0 //TODO: verificar si esta bien este condicional, si es coherente
			THEN
            detener:=1;
            EXIT;
        END_IF
        //muelle
        IF coordxTriangulo<=(nroHorizContMuelle+1)*divHoriz+xt_min //efectivamente la trayectoria pasa sobre los contenedores del muelle
			THEN
            columnaCorresponde:=nroHorizContMuelle+k;
            IF columnaCorresponde<=0
				THEN
                detener:=1;
                EXIT;
            ELSIF alturasContMuelle[columnaCorresponde] > (ySeguridadCarro-distVertTrayectoria)
				THEN
                detener:=1;
                EXIT;
            END_IF
        END_IF
    END_IF
END_FOR
colisionMuelleAlBarcoDesacel:=detener;

END_FUNCTION

// Device/Application/determinarAlturasContenedores
FUNCTION_BLOCK determinarAlturasContenedores
VAR_INPUT
	altoCont: LREAL;
	y_min: LREAL;
END_VAR
VAR_OUTPUT
	alturasContMuelle: ARRAY [1..nroHorizContMuelle] OF LREAL;
	alturasContBarco: ARRAY [1..nroHorizContBarco] OF LREAL;
END_VAR
VAR
	i: INT;
	j: INT;
	cantidadCont: LREAL;
	alturaActual: LREAL;
END_VAR
VAR CONSTANT
	nroHorizContBarco: INT:= 13;
	nroVertContBarco: INT:= 21;
	nroHorizContMuelle: INT:= 7;
	nroVertContMuelle: INT:= 2;
END_VAR

//determinar el perfil de alturas de contenedores y el nro de
//contenedores en cada columna

//barco
FOR i:=1 TO nroHorizContBarco
	DO
	alturasContBarco[i]:=0;
END_FOR
cantidadCont:=0;
FOR j:=1 TO nroHorizContBarco
    //determinar la altura del contenedor actual
    //TODO:mover cantidadCont=0; a esta linea
	DO
    FOR i:=1 TO nroVertContBarco
		DO
        IF contBarco[i,j]=1
			THEN
            cantidadCont:=nroVertContBarco-i+1;
            EXIT;
        END_IF
    END_FOR
    alturaActual:=cantidadCont*altoCont+y_min;
	alturasContBarco[j]:=alturaActual;
END_FOR
// muelle
FOR j:=1 TO nroHorizContMuelle
	DO
    cantidadCont:=0;
    //determinar la altura del contenedor actual
    FOR i:=1 TO nroVertContMuelle
		DO
        IF contMuelle[i,j]=1
			THEN
            cantidadCont:=nroVertContMuelle-i+1;
			EXIT;
        END_IF
    END_FOR
    alturaActual:=cantidadCont*altoCont;
    alturasContMuelle[j]:=alturaActual;
END_FOR

END_FUNCTION_BLOCK

// Device/Application/ControlAngulo
FUNCTION_BLOCK ControlAngulo
VAR_INPUT
	lh: LREAL;
	ml: LREAL;
	TitaMedido: LREAL;
END_VAR
VAR_OUTPUT
	Vtita: LREAL;
END_VAR
VAR
	Derivador1: Derivador;
	Ma: LREAL;
	baa: LREAL;
	Ksaa: LREAL;
	wa: LREAL;
	wposa: LREAL;
	Error: LREAL;
END_VAR
VAR CONSTANT
	g: LREAL:= 9.80665;
	na: LREAL:= 3;
	mc: LREAL:= 50000;
	Mt: LREAL:= 59008;
	Escalado: LREAL:= -2/(3E6);
END_VAR

//Calculo de Ganancias
Ma:= (ml+Mt)/(mc+ml)*lh;
wa:=SQRT(4*(Mt+ml)*Mt*g*lh)/(2*(Mt+ml))*lh;
wposa:=1.6*wa;
baa:=Ma*na*wposa;
Ksaa:=baa*wposa;
//PD
Error:=-TitaMedido;
Derivador1(ValorActual:=Error , Paso:=0.01);
Vtita:= (Derivador1.Derivada*baa+Error*Ksaa)*Escalado;

END_FUNCTION_BLOCK

// Device/Application/Derivador
FUNCTION_BLOCK Derivador
VAR_INPUT
	ValorActual: LREAL;
	Paso: LREAL;//:=0.001;
END_VAR
VAR_OUTPUT
	Derivada: LREAL;
END_VAR
VAR
	init: BOOL:=FALSE;
	ValorAnterior: LREAL:= 0;
END_VAR

Derivada:=(ValorActual-ValorAnterior)/Paso;
ValorAnterior:=ValorActual;
IF (init=FALSE)
	THEN
	Derivada:=0;
	init:=TRUE;
END_IF

END_FUNCTION_BLOCK

// Device/Application/Transferencia
FUNCTION Transferencia : LREAL
VAR_INPUT
	dir:LREAL;
	t:LREAL;
	Vtmanual:LREAL;
	Vtauto:LREAL;
	Vhmanual:LREAL;
	Vhauto:LREAL;
END_VAR
VAR_OUTPUT
	Vt:LREAL:=0;
	Vh:LREAL:=0;
END_VAR
VAR
	m: LREAL;
	y1: LREAL;
	yRecta1: LREAL;
	yRecta2: LREAL;
END_VAR


m:= 1.0/5.0*dir;
IF dir=1 THEN
    y1:=0;
ELSIF dir=-1 THEN
    y1:=1;
END_IF
yRecta1:=m*t+y1;
yRecta2:=1-yRecta1;
Vt:=yRecta1*Vtauto+yRecta2*Vtmanual;
Vh:=yRecta1*Vhauto+yRecta2*Vhmanual;

END_FUNCTION

// Device/Application/rectaDosPuntos
FUNCTION rectaDosPuntos : LREAL
VAR_INPUT
	y2 : LREAL;
	y1 : LREAL;
	x2 : LREAL;
	x1 : LREAL;
	x : LREAL;
END_VAR
VAR
	m: LREAL;
END_VAR

VAR_OUTPUT
	yRecta: LREAL;
END_VAR

m:=(y2-y1)/(x2-x1);
yRecta:=m*(x-x1)+y1;

END_FUNCTION

// Device/Application/nivel2prueba
PROGRAM nivel2prueba
VAR
	PIDl: PIDIzaje;
	PIDt: PIDCarro;
	
	Derivadorl: Derivador;
	Derivadort: Derivador;
	ControlTita: ControlAngulo;
	Saturacionl: Saturation;
	Saturaciont: Saturation;
	RateLimiterl: RateLimiter;
	RateLimitert: RateLimiter;
	ConsignaPos: LREAL;
	ConstPosicion: LREAL:= 2e-1;
END_VAR
VAR CONSTANT
	Bias: LREAL:= -0.245166250000000;
	
END_VAR

//Izaje
Saturacionl(Limite:=vmaxh , Entrada:=vh);
RateLimiterl(Limite:=amaxh , Entrada:=Saturacionl.Salida);
Derivadorl(ValorActual:=lh , Paso:=dt_control);
IF (FuncionamientoIzaje=TRUE)
	THEN
	PIDl(vhConsigna:=RateLimiterl.Salida , vhMedido:=Derivadorl.Derivada);
	ELSE
	PIDl(vhConsigna:=ConsignaIzaje , vhMedido:=Derivadorl.Derivada);
END_IF
Th:=PIDl.th+Bias*ml;
//CARRO
ControlTita(lh:=lh , ml:=ml , TitaMedido:=theta);
IF (ControlPos=TRUE)
	THEN
	ConsignaPos:= (x_destino-xt)*ConstPosicion;
	ELSE
	ConsignaPos:= 0;
END_IF
IF (ControlAngulo=TRUE)
	THEN
	Saturaciont(Limite:=vmaxt , Entrada:=AjusteBordesCarro(xt,AjusteGananciasCarro(vt,ControlTita.Vtita,theta,lh))+ConsignaPos);
ELSE
	Saturaciont(Limite:=vmaxt , Entrada:=AjusteBordesCarro(xt,AjusteGananciasCarro(vt,0,theta,lh))+ConsignaPos);
END_IF
RateLimitert(Limite:=amaxt , Entrada:=Saturaciont.Salida);
Derivadort(ValorActual:=xt , Paso:=dt_control);
IF (FuncionamientoCarro=TRUE)
	THEN
	PIDt(vtConsigna:=RateLimitert.Salida , vtMedido:=Derivadort.Derivada);
	ELSE
	PIDt(vtConsigna:=ConsignaCarro , vtMedido:=Derivadort.Derivada);
END_IF
Tt:=PIDt.tt;
// recordar cambiar los tiempos en derivadores e integradores

END_PROGRAM

// Device/Application/AjusteBordesCarro
FUNCTION AjusteBordesCarro : LREAL
VAR_INPUT
	Xt: LREAL;
	Vt: LREAL;
END_VAR
VAR
	m: LREAL;
	yRecta: LREAL;
END_VAR
VAR CONSTANT
	distanciaSegMaxCarro: LREAL:= 38;
	distanciaSegMinCarro: LREAL:= -18;
	xt_max: LREAL:= 50;
	xt_min: LREAL:= -30;
END_VAR

IF  (Xt<distanciaSegMinCarro AND Vt<0)
	THEN
    m:=1/(distanciaSegMinCarro-xt_min);
    yRecta:=m*(Xt-xt_min);
    IF (yRecta<0)
		THEN
        yRecta:=0;
    END_IF
    Vt:=yRecta*Vt;
END_IF
IF (xt>distanciaSegMaxCarro AND Vt>0)
    THEN
	m:=1/(distanciaSegMaxCarro-xt_max);
    yRecta:=m*(Xt-xt_max);
    IF yRecta<0
		THEN
        yRecta:=0;
    END_IF
    Vt:=yRecta*Vt;
END_IF
AjusteBordesCarro:=Vt;

END_FUNCTION

// Device/Application/AjusteGananciasCarro
FUNCTION AjusteGananciasCarro : LREAL
VAR_INPUT
	VNivel1: LREAL;
	VTita: LREAL;
	tita: LREAL;
	Lh: LREAL;
END_VAR
VAR
	x0: LREAL;
	x1: LREAL;
	x: LREAL;
	m: LREAL;
	y: LREAL;
	Vt: LREAL;
END_VAR
VAR CONSTANT
	pi: LREAL:= 3.141592653589793;
END_VAR

x:=ABS(tita*180/pi);
Vt:=Vnivel1;
IF lh>15
	THEN
    x0:=0;
    x1:=20;
    m:=1/(x1-x0);
    y:=m*(x-x0);
    Vt:=Vtita*y+Vnivel1*(1-y);
END_IF	
IF lh<=15
	THEN
    Vt:=Vtita*30+Vnivel1;
END_IF
AjusteGananciasCarro:=Vt;

END_FUNCTION

// Device/Application/PIDIzaje
FUNCTION_BLOCK PIDIzaje
VAR_INPUT
	vhConsigna: LREAL;
	vhMedido: LREAL;
END_VAR
VAR_OUTPUT
	th: LREAL;
END_VAR
VAR
	Error: LREAL:= 0;
	bah: LREAL:= 57600;
	Ksah: LREAL:= 3.454976303317536E+04;
	Kisah: LREAL:= 1.036185872958829E+04;
	Multiplicador: LREAL:= 1.2;
	Integrador1: Integrador;
	Integrador2: Integrador;
END_VAR

Error:=vhConsigna-vhMedido;
Integrador1(ValorActual:=Error , Paso:=dt_control);
Integrador2(ValorActual:=Integrador1.Integral , Paso:=dt_control);
th:=Error*bah*Multiplicador+Integrador1.Integral*Ksah*EXPT(Multiplicador,2)+Integrador2.Integral*Kisah*EXPT(Multiplicador,3);

END_FUNCTION_BLOCK

// Device/Application/PIDCarro
FUNCTION_BLOCK PIDCarro
VAR_INPUT
	vtConsigna:LREAL;
	vtMedido:LREAL;
END_VAR
VAR_OUTPUT
	tt:LREAL;
END_VAR
VAR
	Error: LREAL:= 0;
	bat: LREAL:= 54000;
	Ksat: LREAL:= 2.470851409978308E+04;
	Kisat: LREAL:= 5.652876564992399E+03;
	Multiplicador: LREAL:= 1.2;
	Integrador1: Integrador;
	Integrador2: Integrador;
END_VAR

Error:=vtConsigna-vtMedido;
Integrador1(ValorActual:=Error , Paso:=dt_control);
Integrador2(ValorActual:=Integrador1.Integral , Paso:=dt_control);
tt:=Error*bat*Multiplicador+Integrador1.Integral*Ksat*EXPT(Multiplicador,2)+Integrador2.Integral*EXPT(Multiplicador,3);

END_FUNCTION_BLOCK

// Device/Application/Saturation
FUNCTION_BLOCK Saturation
VAR_INPUT
	Limite: LREAL;
	Entrada: LREAL;
END_VAR
VAR_OUTPUT
	Salida: LREAL;
END_VAR
VAR
END_VAR

Salida:=Entrada;
IF Entrada>Limite
	THEN Salida:=Limite;
END_IF
IF Entrada<-Limite
	THEN Salida:=-Limite;
END_IF

END_FUNCTION_BLOCK

// Device/Application/RateLimiter
FUNCTION_BLOCK RateLimiter
VAR_INPUT
	Limite: LREAL;
	Entrada: LREAL;
END_VAR
VAR_OUTPUT
	Salida: LREAL;
END_VAR
VAR
	Derivador1: Derivador;
	ValorAnterior: LREAL:= 0;
END_VAR
VAR CONSTANT
	Paso: LREAL:=0.01;
END_VAR

Derivador1(ValorActual:=Entrada , Paso:=0.01);


IF Derivador1.Derivada>Limite
	THEN Salida:=ValorAnterior+Limite*Paso;
	Derivador1(ValorActual:=Salida);
ELSIF Derivador1.Derivada<-Limite
	THEN Salida:=ValorAnterior-Limite*Paso;
	Derivador1(ValorActual:=Salida);
ELSE
		Salida:=Entrada;
END_IF

ValorAnterior:= Salida;

END_FUNCTION_BLOCK

// Device/Application/Planta
PROGRAM Planta
VAR
	Planta_Carro : Carro;
	Planta_Izaje : Izaje;
	Planta_CargaSuspendida : CargaSuspendida;
	Planta_CableElastico : CableElastico; 
END_VAR

Planta_CableElastico(Lh:= Planta_Izaje.Lh , l:= Planta_CargaSuspendida.l , vl:= Planta_Izaje.vl);
Planta_CargaSuspendida(Gancho:= Gcierre , Fw:= Planta_CableElastico.Fw , x:= Planta_Carro.x);
Planta_Carro(SenoCarga:= Planta_CargaSuspendida.Sn , Fw:= Planta_CableElastico.Fw , T:= Tt);
Planta_Izaje(Fw:= Planta_CableElastico.Fw , T:= Th);

xt:= Planta_Carro.x;
ml:= Planta_CargaSuspendida.m;
theta:= ASIN(Planta_CargaSuspendida.Sn);
lh:= Planta_Izaje.Lh;

END_PROGRAM

// Device/Application/CargaSuspendida
FUNCTION_BLOCK CargaSuspendida
VAR_INPUT
	Gancho: bool;
	Fw: LREAL;
	x: LREAL;
END_VAR
VAR_OUTPUT
	m : LREAL:= 17000;
	yl : LREAL:= 39.918277916666670;
	xl : LREAL:= -30;
	l : LREAL:= 5.081722083333332;
	Sn : LREAL:= 0;
END_VAR
VAR
	init: BOOL:= FALSE;
	Integradorx1: Integrador;
	Integradorx2: Integrador;
	Integradory1: Integrador;
	Integradory2: Integrador;
	Cs: LREAL;
END_VAR
VAR CONSTANT
	yt0: LREAL:= 45;
	g: LREAL:= 9.80665;
END_VAR

IF (init=FALSE)
	THEN
	Integradorx2(ValorActual:= -30/dt_planta,Paso:=dt_planta);
	Integradory2(ValorActual:= 39.918277916666670/dt_planta,Paso:=dt_planta);
	init:=TRUE;
END_IF
IF Gancho	THEN
	m:=65000;
	ELSE
	m:=15000;
END_IF
l:= SQRT(EXPT(Integradorx2.Integral-x,2)+EXPT(-Integradory2.Integral+yt0,2));
Cs:= (-Integradory2.Integral+yt0)/l;
Sn:= (Integradorx2.Integral-x)/l;
Integradory1(ValorActual:= Cs*Fw/m-g,Paso:=dt_planta);
Integradory2(ValorActual:= Integradory1.Integral,Paso:=dt_planta);
Integradorx1(ValorActual:= -Sn*Fw/m,Paso:=dt_planta);
Integradorx2(ValorActual:= Integradorx1.Integral,Paso:=dt_planta);

END_FUNCTION_BLOCK

// Device/Application/CableElastico
FUNCTION_BLOCK CableElastico
VAR_INPUT
	Lh: LREAL;
	l: LREAL;
	vl: LREAL;
END_VAR
VAR_OUTPUT
	Fw : LREAL;
END_VAR
VAR
	Derivador1: Derivador;
END_VAR
VAR CONSTANT
	Kw: LREAL:= 1800000;
	bw: LREAL:= 30000;
END_VAR

Derivador1(ValorActual:= l,Paso:=dt_planta);
Fw:= (l-Lh)*Kw+(Derivador1.Derivada-vl)*bw;

END_FUNCTION_BLOCK

// Device/Application/Nivel2
PROGRAM Nivel2
VAR
	PIDl: PIDIzaje;
	PIDt: PIDCarro;
	Derivadorl: Derivador;
	Derivadort: Derivador;
	ControlTita: ControlAngulo;
	Saturacionl: Saturation;
	Saturaciont: Saturation;
	RateLimiterl: RateLimiter;
	RateLimitert: RateLimiter;
	ConsignaPos: LREAL;
	ConstPosicion: LREAL:= 3E-1;
END_VAR
VAR CONSTANT
	Bias: LREAL:= -0.245166250000000;
	
END_VAR

//Izaje
Saturacionl(Limite:=vmaxh , Entrada:=vh);
RateLimiterl(Limite:=amaxh , Entrada:=Saturacionl.Salida);
Derivadorl(ValorActual:=lh , Paso:=0.01);
IF (FuncionamientoIzaje=TRUE)
	THEN
	PIDl(vhConsigna:=RateLimiterl.Salida , vhMedido:=Derivadorl.Derivada);
	ELSE
	PIDl(vhConsigna:=ConsignaIzaje , vhMedido:=Derivadorl.Derivada);
END_IF
Th:=PIDl.th+Bias*ml;
//CARRO
ControlTita(lh:=lh , ml:=ml , TitaMedido:=theta);
IF (ControlPos=TRUE)
	THEN
	ConsignaPos:= (x_destino-xt)*ConstPosicion;
	ELSE
	ConsignaPos:= 0;
END_IF
IF (ControlAngulo=TRUE)
	THEN
	Saturaciont(Limite:=vmaxt , Entrada:=AjusteBordesCarro(xt,AjusteGananciasCarro(vt,ControlTita.Vtita,theta,lh))+ConsignaPos);
ELSE
	Saturaciont(Limite:=vmaxt , Entrada:=AjusteBordesCarro(xt,AjusteGananciasCarro(vt,0,theta,lh))+ConsignaPos);
END_IF
RateLimitert(Limite:=amaxt , Entrada:=Saturaciont.Salida);
Derivadort(ValorActual:=xt , Paso:=0.01);
IF (FuncionamientoCarro=TRUE)
	THEN
	PIDt(vtConsigna:=RateLimitert.Salida , vtMedido:=Derivadort.Derivada);
	ELSE
	PIDt(vtConsigna:=ConsignaCarro , vtMedido:=Derivadort.Derivada);
END_IF
Tt:=PIDt.tt;
// recordar cambiar los tiempos en derivadores e integradores

END_PROGRAM

// Device/Application/Visualization
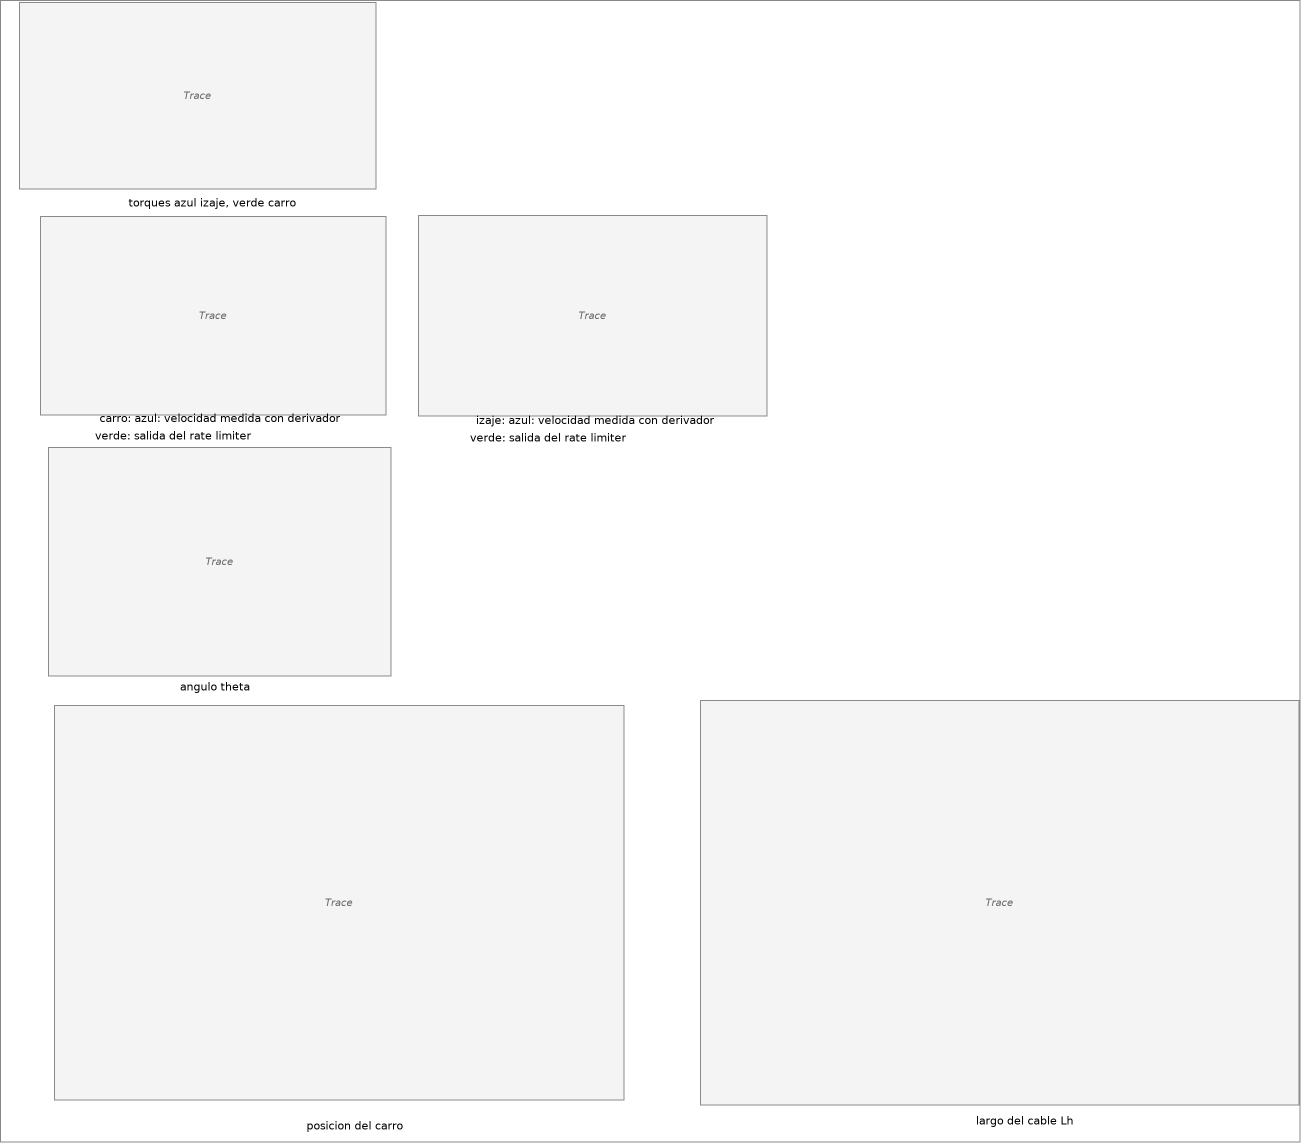
VISUALIZATION Visualization  // 1301x1143
    Trace (40,216 346x199)
    Trace (48,447 343x229)
    Trace (19,2 357x187)
    Label (113,188 199x30), "torques azul izaje, verde carro"
    Label (140,672 150x30), "angulo theta"
    Label (98,421 150x30), "verde: salida del rate limiter"
    Label (81,402 278x33), "carro: azul: velocidad medida con derivador"
    Trace (418,215 349x201)
    Label (456,404 278x33), "izaje: azul: velocidad medida con derivador"
    Label (473,423 150x30), "verde: salida del rate limiter"
    Trace (54,705 570x395)
    Label (280,1111 150x30), "posicion del carro"
    Label (950,1106 150x30), "largo del cable Lh"
    Trace (700,700 599x405)
END_VISUALIZATION
